C01819=1076.283,415.651,391.048,176.432,32.425,155.839
C01820=1076.291,415.898,391.005,176.438,32.436,155.841
C01821=1076.298,416.143,390.962,176.442,32.446,155.843
C01822=1076.305,416.389,390.920,176.447,32.456,155.846
C01823=1076.313,416.636,390.876,176.453,32.466,155.848
C01824=1076.320,416.882,390.833,176.458,32.477,155.850
C01825=1076.327,417.128,390.790,176.463,32.487,155.853
C01826=1076.334,417.374,390.747,176.469,32.497,155.855
C01827=1076.342,417.620,390.703,176.474,32.507,155.857
C01828=1076.349,417.867,390.660,176.480,32.518,155.859
C01829=1076.356,418.112,390.617,176.485,32.529,155.862
C01830=1076.363,418.358,390.574,176.489,32.539,155.864
C01831=1076.371,418.605,390.530,176.495,32.549,155.867
C01832=1076.378,418.850,390.487,176.500,32.560,155.869
C01833=1076.386,419.097,390.443,176.506,32.571,155.871
C01834=1076.392,419.343,390.400,176.511,32.581,155.874
C01835=1076.400,419.589,390.356,176.517,32.592,155.876
C01836=1076.408,419.835,390.312,176.522,32.602,155.879
C01837=1076.415,420.081,390.269,176.528,32.613,155.881
C01838=1076.423,420.327,390.225,176.533,32.624,155.883
C01839=1076.430,420.573,390.182,176.539,32.635,155.886
C01840=1076.438,420.819,390.139,176.544,32.645,155.888
C01841=1076.446,421.066,390.095,176.550,32.656,155.891
C01842=1076.453,421.311,390.051,176.555,32.667,155.893
C01843=1076.460,421.557,390.007,176.561,32.677,155.896
C01844=1076.468,421.804,389.963,176.566,32.688,155.898
C01845=1076.475,422.049,389.920,176.572,32.700,155.901
C01846=1076.482,422.295,389.875,176.577,32.710,155.903
C01847=1076.490,422.542,389.831,176.583,32.721,155.906
C01848=1076.498,422.787,389.787,176.589,32.733,155.908
C01849=1076.505,423.034,389.743,176.594,32.744,155.911
C01850=1076.513,423.279,389.699,176.600,32.755,155.913
C01851=1076.520,423.525,389.656,176.605,32.766,155.916
C01852=1076.527,423.771,389.611,176.611,32.777,155.918
C01853=1076.535,424.017,389.567,176.617,32.789,155.921
C01854=1076.542,424.263,389.522,176.622,32.800,155.924
C01855=1076.550,424.508,389.478,176.628,32.811,155.926
C01856=1076.557,424.755,389.434,176.634,32.823,155.929
C01857=1076.565,425.001,389.390,176.639,32.834,155.931
C01858=1076.573,425.247,389.345,176.645,32.845,155.934
C01859=1076.580,425.493,389.300,176.651,32.857,155.937
C01860=1076.588,425.738,389.256,176.656,32.868,155.939
C01861=1076.595,425.984,389.212,176.662,32.879,155.942
C01862=1076.604,426.253,389.164,176.668,32.892,155.945
C01863=1076.612,426.521,389.115,176.675,32.905,155.948
C01864=1076.620,426.788,389.066,176.681,32.917,155.951
C01865=1076.629,427.057,389.017,176.687,32.930,155.953
C01866=1076.636,427.303,388.973,176.693,32.942,155.956
C01867=1076.644,427.548,388.928,176.699,32.954,155.959
C01868=1076.652,427.794,388.883,176.705,32.965,155.962
C01869=1076.660,428.040,388.839,176.711,32.977,155.964
C01870=1076.667,428.286,388.794,176.717,32.989,155.967
C01871=1076.674,428.532,388.749,176.723,33.001,155.970
C01872=1076.682,428.778,388.703,176.729,33.013,155.973
C01873=1076.690,429.023,388.659,176.735,33.024,155.975
C01874=1076.697,429.270,388.614,176.740,33.037,155.978
C01875=1076.705,429.515,388.568,176.746,33.048,155.981
C01876=1076.713,429.761,388.524,176.753,33.061,155.984
C01877=1076.721,430.006,388.478,176.759,33.073,155.987
C01878=1076.728,430.252,388.434,176.765,33.085,155.989
C01879=1076.736,430.498,388.388,176.771,33.097,155.992
C01880=1076.744,430.744,388.343,176.777,33.109,155.995
C01881=1076.752,430.989,388.298,176.783,33.122,155.998
C01882=1076.760,431.235,388.252,176.790,33.134,156.001
C01883=1076.767,431.481,388.207,176.796,33.146,156.004
C01884=1076.775,431.726,388.162,176.802,33.159,156.007
C01885=1076.784,431.972,388.116,176.808,33.171,156.010
C01886=1076.791,432.218,388.071,176.814,33.184,156.013
C01887=1076.799,432.464,388.025,176.820,33.196,156.015
C01888=1076.806,432.709,387.980,176.826,33.209,156.018
C01889=1076.814,432.955,387.934,176.832,33.221,156.021
C01890=1076.822,433.201,387.888,176.839,33.234,156.024
C01891=1076.830,433.446,387.842,176.846,33.247,156.027
C01892=1076.837,433.692,387.797,176.852,33.259,156.030
C01893=1076.845,433.937,387.751,176.858,33.272,156.033
C01894=1076.853,434.183,387.705,176.865,33.285,156.036
C01895=1076.861,434.429,387.659,176.871,33.298,156.040
C01896=1076.869,434.673,387.613,176.877,33.311,156.043
C01897=1076.877,434.920,387.567,176.883,33.323,156.046
C01898=1076.885,435.165,387.521,176.890,33.337,156.049
C01899=1076.892,435.410,387.476,176.896,33.349,156.052
C01900=1076.901,435.656,387.429,176.902,33.363,156.055
C01901=1076.909,435.901,387.383,176.910,33.376,156.058
C01902=1076.917,436.147,387.337,176.916,33.389,156.061
C01903=1076.925,436.392,387.291,176.922,33.402,156.064
C01904=1076.932,436.639,387.244,176.929,33.415,156.067
C01905=1076.940,436.884,387.198,176.935,33.429,156.071
C01906=1076.948,437.130,387.152,176.943,33.442,156.074
C01907=1076.956,437.374,387.106,176.949,33.455,156.077
C01908=1076.965,437.620,387.059,176.955,33.468,156.080
C01909=1076.973,437.865,387.013,176.962,33.482,156.083
C01910=1076.981,438.111,386.967,176.969,33.495,156.086
C01911=1076.989,438.356,386.920,176.976,33.509,156.090
C01912=1076.998,438.601,386.873,176.982,33.523,156.093
C01913=1077.005,438.848,386.827,176.988,33.536,156.096
C01914=1077.013,439.093,386.780,176.996,33.550,156.099
C01915=1077.022,439.338,386.734,177.002,33.563,156.103
C01916=1077.030,439.584,386.687,177.009,33.577,156.106
C01917=1077.037,439.829,386.640,177.016,33.591,156.109
C01918=1077.048,440.127,386.582,177.024,33.608,156.113
C01919=1077.057,440.426,386.526,177.033,33.625,156.118
C01920=1077.067,440.725,386.469,177.041,33.642,156.122
C01921=1077.078,441.024,386.411,177.050,33.659,156.126
C01922=1077.086,441.269,386.365,177.056,33.673,156.129
C01923=1077.093,441.515,386.317,177.064,33.688,156.133
C01924=1077.102,441.760,386.270,177.070,33.702,156.136
C01925=1077.110,442.006,386.223,177.078,33.716,156.140
C01926=1077.119,442.250,386.175,177.085,33.730,156.143
C01927=1077.127,442.496,386.128,177.092,33.745,156.147
C01928=1077.135,442.740,386.081,177.099,33.759,156.150
C01929=1077.143,442.986,386.033,177.106,33.773,156.154
C01930=1077.152,443.231,385.986,177.113,33.788,156.157
C01931=1077.159,443.477,385.939,177.121,33.803,156.161
C01932=1077.168,443.722,385.891,177.127,33.817,156.164
C01933=1077.176,443.967,385.843,177.135,33.832,156.168
C01934=1077.185,444.213,385.796,177.143,33.847,156.171
C01935=1077.193,444.458,385.748,177.149,33.861,156.175
C01936=1077.201,444.703,385.700,177.157,33.876,156.179
C01937=1077.210,444.948,385.653,177.164,33.891,156.182
C01938=1077.218,445.193,385.605,177.171,33.906,156.186
C01939=1077.226,445.438,385.557,177.179,33.921,156.190
C01940=1077.235,445.683,385.509,177.186,33.936,156.193
C01941=1077.243,445.928,385.461,177.194,33.951,156.197
C01942=1077.251,446.174,385.413,177.202,33.966,156.201
C01943=1077.259,446.419,385.365,177.209,33.981,156.204
C01944=1077.269,446.664,385.317,177.216,33.996,156.208
C01945=1077.277,446.909,385.269,177.223,34.012,156.212
C01946=1077.285,447.154,385.221,177.230,34.027,156.216
C01947=1077.293,447.399,385.173,177.237,34.042,156.219
C01948=1077.303,447.644,385.124,177.242,34.057,156.223
C01949=1077.311,447.890,385.076,177.248,34.072,156.227
C01950=1077.320,448.134,385.027,177.254,34.087,156.231
C01951=1077.329,448.379,384.980,177.260,34.103,156.235
C01952=1077.337,448.624,384.931,177.265,34.117,156.238
C01953=1077.345,448.869,384.883,177.270,34.133,156.242
C01954=1077.355,449.113,384.836,177.275,34.147,156.246
C01955=1077.367,449.358,384.789,177.280,34.161,156.249
C01956=1077.380,449.603,384.743,177.284,34.174,156.253
C01957=1077.394,449.849,384.697,177.288,34.187,156.256
C01958=1077.034,449.844,384.465,177.267,34.346,156.298
C01959=1077.019,449.599,384.511,177.263,34.333,156.295
C01960=1077.006,449.354,384.556,177.258,34.320,156.291
C01961=1076.995,449.108,384.603,177.253,34.306,156.288
C01962=1076.985,448.864,384.651,177.248,34.292,156.284
C01963=1076.976,448.619,384.698,177.243,34.277,156.280
C01964=1076.967,448.374,384.748,177.237,34.261,156.277
C01965=1076.959,448.130,384.796,177.232,34.246,156.273
C01966=1076.949,447.885,384.844,177.226,34.231,156.269
C01967=1076.941,447.640,384.893,177.220,34.216,156.265
C01968=1076.933,447.395,384.941,177.213,34.201,156.261
C01969=1076.924,447.150,384.990,177.206,34.185,156.258
C01970=1076.916,446.904,385.038,177.199,34.170,156.254
C01971=1076.907,446.660,385.085,177.192,34.156,156.250
C01972=1076.899,446.415,385.134,177.185,34.140,156.246
C01973=1076.891,446.170,385.182,177.177,34.125,156.243
C01974=1076.881,445.924,385.230,177.170,34.110,156.239
C01975=1076.873,445.679,385.278,177.162,34.095,156.235
C01976=1076.865,445.434,385.326,177.155,34.080,156.231
C01977=1076.857,445.189,385.375,177.147,34.065,156.228
C01978=1076.848,444.944,385.422,177.139,34.050,156.224
C01979=1076.840,444.699,385.470,177.132,34.035,156.220
C01980=1076.832,444.453,385.517,177.125,34.020,156.217
C01981=1076.823,444.208,385.565,177.117,34.005,156.213
C01982=1076.815,443.963,385.613,177.110,33.991,156.210
C01983=1076.806,443.718,385.660,177.102,33.976,156.206
C01984=1076.798,443.473,385.708,177.096,33.962,156.202
C01985=1076.789,443.228,385.755,177.088,33.947,156.199
C01986=1076.781,442.982,385.803,177.081,33.932,156.195
C01987=1076.773,442.737,385.851,177.073,33.918,156.192
C01988=1076.765,442.492,385.898,177.067,33.904,156.188
C01989=1076.756,442.246,385.946,177.059,33.889,156.185
C01990=1076.748,442.001,385.993,177.052,33.875,156.181
C01991=1076.740,441.756,386.041,177.045,33.861,156.178
C01992=1076.732,441.511,386.087,177.038,33.847,156.174
C01993=1076.723,441.265,386.134,177.030,33.833,156.171
C01994=1076.715,441.020,386.182,177.024,33.818,156.168
C01995=1076.706,440.739,386.236,177.015,33.802,156.164
C01996=1076.696,440.456,386.289,177.007,33.786,156.160
C01997=1076.687,440.175,386.344,177.000,33.770,156.156
C01998=1076.678,439.894,386.397,176.991,33.754,156.152
C01999=1076.669,439.649,386.444,176.984,33.740,156.149
C02000=1076.661,439.403,386.491,176.978,33.727,156.145
C02001=1076.653,439.158,386.538,176.970,33.713,156.142
C02002=1076.645,438.912,386.584,176.964,33.699,156.139
C02003=1076.636,438.667,386.631,176.957,33.686,156.136
C02004=1076.628,438.421,386.678,176.950,33.672,156.132
C02005=1076.620,438.176,386.725,176.943,33.658,156.129
C02006=1076.612,437.930,386.771,176.937,33.645,156.126
C02007=1076.604,437.685,386.817,176.930,33.631,156.123
C02008=1076.596,437.440,386.864,176.923,33.618,156.119
C02009=1076.587,437.194,386.911,176.916,33.605,156.116
C02010=1076.580,436.949,386.956,176.910,33.591,156.113
C02011=1076.571,436.703,387.003,176.903,33.578,156.110
C02012=1076.564,436.458,387.049,176.896,33.565,156.107
C02013=1076.556,436.212,387.096,176.889,33.552,156.103
C02014=1076.548,435.967,387.142,176.883,33.538,156.100
C02015=1076.539,435.721,387.188,176.877,33.526,156.097
C02016=1076.532,435.476,387.234,176.870,33.513,156.094
C02017=1076.523,435.230,387.281,176.864,33.499,156.091
C02018=1076.516,434.985,387.326,176.857,33.487,156.088
C02019=1076.508,434.739,387.372,176.850,33.473,156.085
C02020=1076.499,434.494,387.419,176.844,33.461,156.082
C02021=1076.492,434.248,387.464,176.837,33.448,156.079
C02022=1076.484,434.003,387.510,176.831,33.435,156.076
C02023=1076.476,433.757,387.556,176.824,33.422,156.073
C02024=1076.468,433.511,387.602,176.818,33.410,156.070
C02025=1076.461,433.266,387.647,176.812,33.397,156.067
C02026=1076.452,433.020,387.693,176.805,33.384,156.064
C02027=1076.445,432.774,387.739,176.799,33.371,156.061
C02028=1076.437,432.529,387.785,176.793,33.359,156.058
C02029=1076.429,432.283,387.830,176.786,33.346,156.055
C02030=1076.421,432.037,387.876,176.780,33.334,156.052
C02031=1076.414,431.792,387.922,176.774,33.321,156.049
C02032=1076.406,431.546,387.968,176.768,33.309,156.046
C02033=1076.398,431.301,388.012,176.761,33.297,156.043
C02034=1076.390,431.055,388.058,176.755,33.285,156.040
C02035=1076.382,430.809,388.104,176.749,33.272,156.037
C02036=1076.375,430.563,388.149,176.742,33.260,156.034
C02037=1076.366,430.318,388.194,176.736,33.248,156.032
C02038=1076.359,430.073,388.239,176.731,33.236,156.029
C02039=1076.351,429.826,388.284,176.725,33.223,156.026
C02040=1076.344,429.581,388.330,176.719,33.211,156.023
C02041=1076.336,429.335,388.374,176.712,33.199,156.020
C02042=1076.328,429.090,388.420,176.706,33.187,156.017
C02043=1076.320,428.843,388.465,176.700,33.176,156.015
C02044=1076.312,428.597,388.509,176.694,33.163,156.012
C02045=1076.304,428.352,388.555,176.688,33.151,156.009
C02046=1076.297,428.106,388.600,176.682,33.140,156.006
C02047=1076.290,427.860,388.645,176.676,33.128,156.004
C02048=1076.282,427.614,388.689,176.670,33.116,156.001
C02049=1076.274,427.368,388.734,176.664,33.104,155.998
C02050=1076.266,427.122,388.779,176.659,33.092,155.995
C02051=1076.258,426.853,388.828,176.651,33.080,155.993
C02052=1076.249,426.583,388.877,176.645,33.067,155.990
C02053=1076.240,426.314,388.926,176.639,33.054,155.987
C02054=1076.232,426.044,388.975,176.632,33.042,155.984
C02055=1076.225,425.798,389.020,176.627,33.031,155.981
C02056=1076.217,425.552,389.064,176.621,33.019,155.978
C02057=1076.210,425.307,389.109,176.615,33.007,155.976
C02058=1076.202,425.061,389.153,176.609,32.996,155.973
C02059=1076.194,424.814,389.197,176.603,32.985,155.970
C02060=1076.187,424.568,389.241,176.597,32.973,155.968
C02061=1076.179,424.323,389.286,176.592,32.962,155.965
C02062=1076.171,424.077,389.331,176.586,32.951,155.963
C02063=1076.164,423.831,389.374,176.580,32.939,155.960
C02064=1076.157,423.585,389.419,176.575,32.929,155.958
C02065=1076.149,423.339,389.463,176.569,32.917,155.955
C02066=1076.141,423.093,389.507,176.564,32.906,155.952
C02067=1076.134,422.847,389.551,176.558,32.895,155.950
C02068=1076.127,422.601,389.595,176.552,32.884,155.947
C02069=1076.119,422.355,389.639,176.547,32.873,155.945
C02070=1076.112,422.109,389.683,176.540,32.862,155.942
C02071=1076.104,421.863,389.727,176.535,32.851,155.940
C02072=1076.096,421.617,389.771,176.529,32.840,155.937
C02073=1076.090,421.371,389.815,176.524,32.829,155.935
C02074=1076.082,421.125,389.859,176.518,32.818,155.932
C02075=1076.074,420.879,389.903,176.513,32.807,155.930
C02076=1076.067,420.634,389.946,176.507,32.797,155.927
C02077=1076.059,420.387,389.990,176.502,32.786,155.925
C02078=1076.051,420.141,390.033,176.496,32.775,155.923
C02079=1076.044,419.895,390.077,176.491,32.764,155.920
C02080=1076.037,419.648,390.121,176.485,32.754,155.918
C02081=1076.030,419.403,390.164,176.480,32.743,155.915
C02082=1076.022,419.156,390.208,176.474,32.733,155.913
C02083=1076.014,418.910,390.251,176.469,32.722,155.911
C02084=1076.007,418.664,390.295,176.463,32.711,155.908
C02085=1076.000,418.418,390.338,176.458,32.701,155.906
C02086=1075.992,418.172,390.382,176.453,32.691,155.903
C02087=1075.985,417.926,390.425,176.447,32.680,155.901
C02088=1075.977,417.680,390.468,176.442,32.670,155.899
C02089=1075.970,417.434,390.512,176.436,32.660,155.896
C02090=1075.963,417.188,390.555,176.431,32.649,155.894
C02091=1075.956,416.942,390.598,176.426,32.639,155.892
C02092=1075.948,416.696,390.641,176.421,32.628,155.889
C02093=1075.941,416.450,390.685,176.416,32.618,155.887
C02094=1075.933,416.203,390.728,176.411,32.608,155.885
C02095=1075.926,415.957,390.771,176.405,32.598,155.882
C02096=1075.919,415.712,390.814,176.400,32.587,155.880
C02097=1075.911,415.465,390.857,176.395,32.578,155.878
C02098=1075.904,415.219,390.900,176.389,32.567,155.876
C02099=1075.897,414.973,390.943,176.384,32.557,155.873
C02100=1075.890,414.726,390.986,176.379,32.547,155.871
C02101=1075.882,414.480,391.028,176.374,32.537,155.869
C02102=1075.875,414.234,391.071,176.368,32.527,155.867
C02103=1075.867,413.988,391.115,176.363,32.517,155.864
C02104=1075.861,413.741,391.157,176.358,32.507,155.862
C02105=1075.853,413.495,391.199,176.354,32.497,155.860
C02106=1075.845,413.249,391.243,176.348,32.487,155.858
C02107=1075.838,412.997,391.286,176.343,32.478,155.856
C02108=1075.831,412.745,391.329,176.338,32.468,155.853
C02109=1075.823,412.493,391.373,176.332,32.458,155.851
C02110=1075.816,412.241,391.417,176.327,32.448,155.849
C02111=1075.809,411.995,391.459,176.322,32.438,155.847
C02112=1075.801,411.749,391.501,176.317,32.429,155.845
C02113=1075.794,411.502,391.544,176.312,32.419,155.842
C02114=1075.787,411.255,391.587,176.307,32.409,155.840
C02115=1075.779,411.010,391.629,176.302,32.399,155.838
C02116=1075.773,410.763,391.671,176.297,32.390,155.836
C02117=1075.766,410.517,391.714,176.292,32.380,155.834
C02118=1075.758,410.271,391.756,176.287,32.371,155.832
C02119=1075.751,410.025,391.798,176.282,32.361,155.830
C02120=1075.744,409.778,391.841,176.277,32.352,155.828
C02121=1075.736,409.532,391.883,176.272,32.342,155.826
C02122=1075.730,409.285,391.925,176.267,32.333,155.823
C02123=1075.722,409.039,391.967,176.262,32.323,155.821
C02124=1075.715,408.793,392.009,176.257,32.314,155.819
C02125=1075.708,408.546,392.052,176.252,32.305,155.817
C02126=1075.701,408.300,392.093,176.247,32.295,155.815
C02127=1075.694,408.053,392.136,176.243,32.286,155.813
C02128=1075.687,407.807,392.178,176.238,32.276,155.811
C02129=1075.680,407.561,392.219,176.233,32.268,155.809
C02130=1075.673,407.314,392.262,176.228,32.258,155.807
C02131=1075.667,407.068,392.303,176.223,32.249,155.805
C02132=1075.660,406.822,392.345,176.219,32.240,155.803
C02133=1075.652,406.575,392.387,176.214,32.230,155.801
C02134=1075.645,406.329,392.429,176.209,32.221,155.799
C02135=1075.638,406.083,392.470,176.204,32.213,155.797
C02136=1075.631,405.837,392.512,176.199,32.203,155.795
C02137=1075.624,405.590,392.554,176.195,32.194,155.793
C02138=1075.617,405.343,392.595,176.190,32.185,155.791
C02139=1075.609,405.097,392.637,176.185,32.176,155.789
C02140=1075.603,404.850,392.679,176.180,32.167,155.787
C02141=1075.595,404.604,392.720,176.175,32.158,155.785
C02142=1075.589,404.358,392.761,176.171,32.149,155.783
C02143=1075.582,404.111,392.804,176.166,32.141,155.781
C02144=1075.575,403.865,392.845,176.162,32.132,155.779
C02145=1075.567,403.618,392.886,176.157,32.123,155.777
C02146=1075.560,403.372,392.927,176.152,32.114,155.775
C02147=1075.554,403.125,392.969,176.148,32.105,155.774
C02148=1075.547,402.879,393.010,176.143,32.096,155.772
C02149=1075.539,402.632,393.051,176.138,32.088,155.770
C02150=1075.532,402.386,393.093,176.133,32.079,155.768
C02151=1075.525,402.139,393.134,176.129,32.070,155.766
C02152=1075.518,401.893,393.175,176.124,32.062,155.764
C02153=1075.512,401.646,393.216,176.120,32.053,155.762
C02154=1075.504,401.400,393.258,176.115,32.044,155.760
C02155=1075.498,401.154,393.299,176.111,32.035,155.759
C02156=1075.490,400.907,393.340,176.106,32.027,155.757
C02157=1075.483,400.661,393.381,176.101,32.019,155.755
C02158=1075.477,400.414,393.421,176.096,32.010,155.753
C02159=1075.470,400.179,393.461,176.093,32.002,155.751
C02160=1075.464,399.943,393.500,176.088,31.994,155.750
C02161=1075.456,399.708,393.539,176.084,31.986,155.748
C02162=1075.450,399.472,393.578,176.079,31.978,155.746
C02163=1075.443,399.237,393.618,176.075,31.970,155.744
C02164=1075.437,399.001,393.657,176.071,31.961,155.743
C02165=1075.430,398.765,393.695,176.066,31.953,155.741
C02166=1075.421,398.432,393.750,176.060,31.942,155.738
C02167=1075.414,398.186,393.791,176.056,31.934,155.737
C02168=1075.407,397.939,393.832,176.051,31.925,155.735
C02169=1075.400,397.692,393.873,176.047,31.917,155.733
C02170=1075.393,397.446,393.913,176.043,31.909,155.731
C02171=1075.386,397.199,393.954,176.038,31.901,155.730
C02172=1075.380,396.953,393.994,176.033,31.892,155.728
C02173=1075.372,396.706,394.036,176.029,31.885,155.726
C02174=1075.366,396.460,394.076,176.025,31.876,155.724
C02175=1075.358,396.213,394.116,176.020,31.868,155.723
C02176=1075.351,395.967,394.157,176.015,31.860,155.721
C02177=1075.345,395.720,394.197,176.012,31.852,155.719
C02178=1075.338,395.473,394.237,176.007,31.844,155.717
C02179=1075.331,395.227,394.278,176.002,31.835,155.716
C02180=1075.324,394.980,394.319,175.998,31.827,155.714
C02181=1075.317,394.734,394.358,175.994,31.819,155.712
C02182=1075.311,394.487,394.398,175.989,31.811,155.711
C02183=1075.304,394.240,394.439,175.985,31.803,155.709
C02184=1075.297,393.994,394.480,175.981,31.795,155.707
C02185=1075.290,393.747,394.520,175.976,31.787,155.705
C02186=1075.283,393.501,394.560,175.972,31.779,155.704
C02187=1075.277,393.254,394.600,175.968,31.772,155.702
C02188=1075.269,393.007,394.640,175.963,31.764,155.701
C02189=1075.263,392.761,394.680,175.959,31.756,155.699
C02190=1075.256,392.514,394.720,175.954,31.748,155.697
C02191=1075.249,392.268,394.760,175.950,31.740,155.695
C02192=1075.242,392.021,394.800,175.946,31.732,155.694
C02193=1075.236,391.774,394.840,175.941,31.724,155.692
C02194=1075.229,391.528,394.880,175.937,31.716,155.691
C02195=1075.222,391.282,394.920,175.933,31.709,155.689
C02196=1075.215,391.034,394.959,175.928,31.701,155.687
C02197=1075.208,390.788,394.999,175.924,31.694,155.686
C02198=1075.201,390.541,395.039,175.920,31.686,155.684
C02199=1075.195,390.295,395.079,175.915,31.678,155.683
C02200=1075.187,390.048,395.119,175.912,31.670,155.681
C02201=1075.181,389.801,395.158,175.907,31.663,155.679
C02202=1075.174,389.555,395.198,175.902,31.655,155.678
C02203=1075.167,389.308,395.237,175.899,31.648,155.676
C02204=1075.161,389.061,395.277,175.894,31.640,155.675
C02205=1075.153,388.814,395.317,175.890,31.633,155.673
C02206=1075.147,388.568,395.357,175.886,31.625,155.671
C02207=1075.140,388.321,395.396,175.881,31.617,155.670
C02208=1075.133,388.075,395.435,175.877,31.610,155.668
C02209=1075.127,387.828,395.475,175.873,31.603,155.667
C02210=1075.120,387.582,395.514,175.869,31.595,155.665
C02211=1075.113,387.335,395.553,175.864,31.588,155.664
C02212=1075.106,387.088,395.593,175.861,31.580,155.662
C02213=1075.100,386.841,395.632,175.856,31.573,155.661
C02214=1075.093,386.595,395.672,175.852,31.565,155.659
C02215=1075.086,386.354,395.710,175.848,31.558,155.658
C02216=1075.080,386.114,395.748,175.844,31.551,155.656
C02217=1075.074,385.874,395.786,175.839,31.544,155.655
C02218=1075.067,385.633,395.825,175.836,31.537,155.653
C02219=1075.060,385.394,395.863,175.832,31.530,155.652
C02220=1075.054,385.153,395.901,175.828,31.522,155.650
C02221=1075.047,384.913,395.940,175.824,31.515,155.649
C02222=1075.041,384.672,395.978,175.819,31.508,155.647
C02223=1075.034,384.425,396.017,175.816,31.501,155.646
C02224=1075.027,384.179,396.056,175.811,31.494,155.644
C02225=1075.021,383.932,396.095,175.807,31.486,155.643
C02226=1075.015,383.686,396.134,175.804,31.479,155.641
C02227=1075.008,383.439,396.173,175.799,31.472,155.640
C02228=1075.001,383.192,396.212,175.795,31.464,155.638
C02229=1074.995,382.945,396.251,175.791,31.457,155.637
C02230=1074.988,382.698,396.290,175.787,31.451,155.635
C02231=1074.981,382.451,396.329,175.782,31.443,155.634
C02232=1074.974,382.204,396.368,175.779,31.436,155.632
C02233=1074.968,381.957,396.407,175.774,31.429,155.631
C02234=1074.962,381.711,396.445,175.771,31.422,155.629
C02235=1074.955,381.464,396.484,175.766,31.415,155.628
C02236=1074.949,381.218,396.523,175.762,31.408,155.627
C02237=1074.942,380.971,396.562,175.759,31.401,155.625
C02238=1074.935,380.724,396.601,175.754,31.394,155.624
C02239=1074.928,380.477,396.640,175.750,31.387,155.622
C02240=1074.922,380.230,396.678,175.746,31.380,155.621
C02241=1074.915,379.983,396.717,175.742,31.373,155.619
C02242=1074.909,379.737,396.755,175.739,31.366,155.618
C02243=1074.902,379.490,396.794,175.734,31.359,155.617
C02244=1074.895,379.243,396.831,175.730,31.352,155.615
C02245=1074.888,378.996,396.870,175.726,31.345,155.614
C02246=1074.881,378.749,396.909,175.722,31.338,155.612
C02247=1074.875,378.502,396.947,175.719,31.332,155.611
C02248=1074.868,378.256,396.986,175.714,31.324,155.610
C02249=1074.862,378.008,397.024,175.710,31.318,155.608
C02250=1074.855,377.761,397.063,175.706,31.311,155.607
C02251=1074.849,377.515,397.101,175.702,31.304,155.605
C02252=1074.842,377.268,397.139,175.698,31.298,155.604
C02253=1074.835,377.021,397.178,175.694,31.291,155.603
C02254=1074.829,376.773,397.216,175.690,31.284,155.601
C02255=1074.823,376.527,397.255,175.687,31.277,155.600
C02256=1074.815,376.280,397.292,175.682,31.270,155.599
C02257=1074.809,376.033,397.330,175.678,31.264,155.597
C02258=1074.803,375.787,397.369,175.675,31.257,155.596
C02259=1074.796,375.539,397.407,175.670,31.250,155.595
C02260=1074.789,375.292,397.446,175.667,31.243,155.593
C02261=1074.783,375.046,397.484,175.663,31.237,155.592
C02262=1074.777,374.798,397.522,175.658,31.230,155.590
C02263=1074.771,374.551,397.559,175.655,31.223,155.589
C02264=1074.764,374.305,397.598,175.651,31.217,155.588
C02265=1074.757,374.057,397.636,175.648,31.210,155.586
C02266=1074.751,373.811,397.674,175.643,31.203,155.585
C02267=1074.745,373.563,397.712,175.639,31.197,155.584
C02268=1074.738,373.317,397.750,175.636,31.191,155.583
C02269=1074.731,373.070,397.788,175.631,31.183,155.581
C02270=1074.725,372.823,397.826,175.628,31.177,155.580
C02271=1074.718,372.597,397.860,175.624,31.171,155.579
C02272=1074.713,372.371,397.895,175.620,31.165,155.578
C02273=1074.707,372.145,397.928,175.617,31.159,155.576
C02274=1074.701,371.920,397.963,175.613,31.153,155.575
C02275=1074.695,371.694,397.998,175.610,31.148,155.574
C02276=1074.689,371.468,398.032,175.607,31.142,155.573
C02277=1074.683,371.243,398.067,175.603,31.136,155.572
C02278=1074.677,371.017,398.102,175.600,31.130,155.570
C02279=1074.670,370.770,398.139,175.596,31.124,155.569
C02280=1074.664,370.523,398.177,175.591,31.117,155.568
C02281=1074.657,370.276,398.213,175.588,31.111,155.567
C02282=1074.651,370.028,398.252,175.584,31.104,155.565
C02283=1074.644,369.782,398.289,175.581,31.098,155.564
C02284=1074.638,369.535,398.327,175.576,31.092,155.563
C02285=1074.631,369.288,398.364,175.572,31.086,155.562
C02286=1074.625,369.041,398.402,175.569,31.079,155.560
C02287=1074.618,368.794,398.439,175.565,31.073,155.559
C02288=1074.612,368.546,398.477,175.562,31.067,155.558
C02289=1074.605,368.300,398.514,175.557,31.060,155.557
C02290=1074.600,368.052,398.551,175.554,31.054,155.555
C02291=1074.592,367.805,398.588,175.550,31.048,155.554
C02292=1074.586,367.559,398.626,175.546,31.041,155.553
C02293=1074.579,367.311,398.663,175.543,31.035,155.552
C02294=1074.574,367.064,398.701,175.538,31.029,155.550
C02295=1074.567,366.818,398.738,175.535,31.023,155.549
C02296=1074.561,366.570,398.775,175.531,31.016,155.548
C02297=1074.554,366.323,398.812,175.527,31.010,155.547
C02298=1074.548,366.076,398.849,175.524,31.004,155.546
C02299=1074.541,365.829,398.887,175.519,30.998,155.544
C02300=1074.536,365.581,398.924,175.516,30.992,155.543
C02301=1074.529,365.335,398.961,175.512,30.985,155.542
C02302=1074.522,365.087,398.998,175.509,30.979,155.541
C02303=1074.516,364.840,399.036,175.505,30.973,155.540
C02304=1074.510,364.593,399.072,175.501,30.967,155.538
C02305=1074.503,364.345,399.109,175.498,30.961,155.537
C02306=1074.497,364.099,399.147,175.493,30.955,155.536
C02307=1074.491,363.852,399.183,175.490,30.949,155.535
C02308=1074.484,363.604,399.220,175.486,30.943,155.534
C02309=1074.477,363.357,399.257,175.483,30.937,155.532
C02310=1074.471,363.110,399.294,175.479,30.931,155.531
C02311=1074.465,362.862,399.331,175.475,30.925,155.530
C02312=1074.458,362.615,399.368,175.472,30.919,155.529
C02313=1074.452,362.368,399.404,175.467,30.913,155.528
C02314=1074.445,362.122,399.441,175.464,30.907,155.527
C02315=1074.438,361.874,399.478,175.460,30.901,155.525
C02316=1074.433,361.627,399.515,175.457,30.895,155.524
C02317=1074.426,361.380,399.551,175.453,30.889,155.523
C02318=1074.420,361.133,399.588,175.449,30.883,155.522
C02319=1074.413,360.885,399.625,175.446,30.877,155.521
C02320=1074.407,360.638,399.661,175.442,30.871,155.520
C02321=1074.400,360.391,399.698,175.439,30.865,155.518
C02322=1074.394,360.144,399.734,175.434,30.859,155.517
C02323=1074.388,359.896,399.771,175.431,30.853,155.516
C02324=1074.382,359.649,399.807,175.427,30.848,155.515
C02325=1074.375,359.401,399.844,175.424,30.842,155.514
C02326=1074.369,359.154,399.881,175.420,30.836,155.513
C02327=1074.363,358.937,399.912,175.417,30.831,155.512
C02328=1074.357,358.720,399.945,175.414,30.826,155.511
C02329=1074.352,358.503,399.976,175.410,30.821,155.510
C02330=1074.346,358.285,400.009,175.407,30.815,155.509
C02331=1074.340,358.068,400.040,175.404,30.810,155.508
C02332=1074.335,357.850,400.072,175.401,30.805,155.507
C02333=1074.329,357.633,400.105,175.398,30.800,155.506
C02334=1074.324,357.416,400.137,175.395,30.795,155.505
C02335=1074.317,357.168,400.173,175.391,30.790,155.504
C02336=1074.311,356.921,400.209,175.387,30.783,155.503
C02337=1074.305,356.674,400.246,175.383,30.778,155.502
C02338=1074.298,356.426,400.282,175.380,30.772,155.501
C02339=1074.292,356.179,400.318,175.376,30.766,155.499
C02340=1074.285,355.932,400.354,175.373,30.760,155.498
C02341=1074.279,355.685,400.390,175.369,30.755,155.497
C02342=1074.273,355.437,400.426,175.366,30.750,155.496
C02343=1074.267,355.190,400.462,175.362,30.744,155.495
C02344=1074.260,354.943,400.499,175.358,30.738,155.494
C02345=1074.254,354.696,400.534,175.355,30.732,155.493
C02346=1074.248,354.448,400.571,175.351,30.727,155.492
C02347=1074.242,354.201,400.607,175.348,30.721,155.491
C02348=1074.236,353.954,400.643,175.344,30.715,155.490
C02349=1074.229,353.706,400.678,175.341,30.710,155.489
C02350=1074.222,353.459,400.715,175.337,30.704,155.488
C02351=1074.216,353.212,400.750,175.334,30.698,155.486
C02352=1074.210,352.965,400.787,175.330,30.693,155.485
C02353=1074.204,352.717,400.823,175.326,30.687,155.484
C02354=1074.198,352.469,400.858,175.323,30.682,155.483
C02355=1074.191,352.223,400.894,175.319,30.676,155.482
C02356=1074.185,351.975,400.930,175.316,30.670,155.481
C02357=1074.179,351.727,400.966,175.312,30.665,155.480
C02358=1074.172,351.480,401.001,175.309,30.659,155.479
C02359=1074.166,351.233,401.037,175.305,30.654,155.478
C02360=1074.160,350.985,401.073,175.302,30.648,155.477
C02361=1074.153,350.738,401.108,175.298,30.643,155.476
C02362=1074.147,350.491,401.144,175.295,30.638,155.475
C02363=1074.141,350.243,401.180,175.292,30.632,155.474
C02364=1074.134,349.996,401.215,175.288,30.627,155.473
C02365=1074.128,349.749,401.251,175.285,30.621,155.472
C02366=1074.122,349.501,401.286,175.281,30.616,155.471
C02367=1074.116,349.254,401.322,175.278,30.610,155.470
C02368=1074.109,349.007,401.358,175.274,30.605,155.469
C02369=1074.102,348.759,401.393,175.271,30.600,155.468
C02370=1074.096,348.511,401.429,175.267,30.594,155.467
C02371=1074.091,348.265,401.464,175.264,30.589,155.466
C02372=1074.084,348.017,401.499,175.260,30.583,155.465
C02373=1074.078,347.769,401.535,175.256,30.578,155.464
C02374=1074.071,347.522,401.570,175.253,30.572,155.463
C02375=1074.065,347.274,401.606,175.249,30.567,155.462
C02376=1074.059,347.027,401.641,175.247,30.562,155.461
C02377=1074.053,346.780,401.676,175.243,30.556,155.460
C02378=1074.046,346.533,401.712,175.240,30.551,155.459
C02379=1074.041,346.284,401.747,175.236,30.545,155.458
C02380=1074.035,346.037,401.782,175.233,30.540,155.457
C02381=1074.029,345.790,401.817,175.229,30.535,155.456
C02382=1074.022,345.543,401.852,175.226,30.529,155.455
C02383=1074.017,345.327,401.883,175.223,30.525,155.454
C02384=1074.011,345.112,401.914,175.219,30.520,155.453
C02385=1074.005,344.896,401.944,175.217,30.516,155.452
C02386=1074.001,344.680,401.975,175.214,30.511,155.451
C02387=1073.995,344.464,402.006,175.211,30.506,155.450
C02388=1073.989,344.249,402.037,175.208,30.502,155.449
C02389=1073.984,344.033,402.067,175.205,30.497,155.449
C02390=1073.979,343.817,402.098,175.202,30.492,155.448
C02391=1073.972,343.570,402.133,175.198,30.487,155.447
C02392=1073.966,343.321,402.168,175.195,30.482,155.446
C02393=1073.960,343.075,402.203,175.192,30.477,155.445
C02394=1073.953,342.827,402.238,175.189,30.472,155.444
C02395=1073.947,342.579,402.272,175.185,30.467,155.443
C02396=1073.941,342.332,402.307,175.181,30.462,155.442
C02397=1073.935,342.084,402.342,175.178,30.456,155.441
C02398=1073.928,341.837,402.377,175.174,30.451,155.440
C02399=1073.922,341.590,402.411,175.171,30.446,155.439
C02400=1073.916,341.342,402.447,175.168,30.441,155.438
C02401=1073.910,341.094,402.481,175.165,30.436,155.437
C02402=1073.904,340.848,402.516,175.161,30.430,155.436
C02403=1073.897,340.600,402.550,175.158,30.425,155.435
C02404=1073.891,340.352,402.586,175.154,30.420,155.434
C02405=1073.885,340.105,402.620,175.152,30.415,155.433
C02406=1073.879,339.857,402.655,175.148,30.410,155.432
C02407=1073.873,339.610,402.689,175.145,30.405,155.432
C02408=1073.867,339.362,402.724,175.141,30.399,155.431
C02409=1073.860,339.114,402.760,175.137,30.394,155.430
C02410=1073.854,338.867,402.794,175.134,30.389,155.429
C02411=1073.848,338.620,402.829,175.131,30.384,155.428
C02412=1073.842,338.372,402.863,175.128,30.379,155.427
C02413=1073.836,338.124,402.898,175.124,30.374,155.426
C02414=1073.830,337.877,402.932,175.121,30.369,155.425
C02415=1073.823,337.629,402.967,175.118,30.364,155.424
C02416=1073.817,337.382,403.001,175.115,30.359,155.423
C02417=1073.811,337.134,403.035,175.111,30.354,155.422
C02418=1073.805,336.886,403.070,175.108,30.349,155.421
C02419=1073.799,336.639,403.104,175.104,30.344,155.420
C02420=1073.792,336.391,403.138,175.102,30.339,155.419
C02421=1073.786,336.144,403.173,175.098,30.334,155.418
C02422=1073.780,335.896,403.208,175.095,30.329,155.418
C02423=1073.774,335.649,403.242,175.091,30.324,155.417
C02424=1073.767,335.401,403.276,175.088,30.319,155.416
C02425=1073.761,335.154,403.310,175.085,30.314,155.415
C02426=1073.755,334.906,403.344,175.081,30.309,155.414
C02427=1073.749,334.658,403.379,175.078,30.304,155.413
C02428=1073.743,334.410,403.413,175.075,30.299,155.412
C02429=1073.737,334.163,403.447,175.072,30.294,155.411
C02430=1073.731,333.916,403.481,175.068,30.289,155.410
C02431=1073.724,333.668,403.515,175.065,30.284,155.409
C02432=1073.719,333.421,403.550,175.062,30.279,155.409
C02433=1073.712,333.173,403.584,175.059,30.274,155.408
C02434=1073.706,332.925,403.618,175.055,30.269,155.407
C02435=1073.700,332.677,403.652,175.052,30.264,155.406
C02436=1073.693,332.430,403.685,175.049,30.260,155.405
C02437=1073.688,332.182,403.719,175.046,30.255,155.404
C02438=1073.681,331.934,403.754,175.042,30.250,155.403
C02439=1073.676,331.716,403.783,175.039,30.245,155.402
C02440=1073.671,331.498,403.814,175.037,30.241,155.402
C02441=1073.666,331.280,403.844,175.034,30.237,155.401
C02442=1073.660,331.062,403.874,175.031,30.232,155.400
C02443=1073.655,330.844,403.904,175.028,30.228,155.399
C02444=1073.649,330.625,403.933,175.025,30.224,155.399
C02445=1073.643,330.407,403.963,175.022,30.219,155.398
C02446=1073.638,330.189,403.992,175.019,30.216,155.397
C02447=1073.631,329.940,404.026,175.016,30.211,155.396
C02448=1073.625,329.693,404.060,175.013,30.206,155.395
C02449=1073.618,329.445,404.094,175.010,30.201,155.395
C02450=1073.613,329.198,404.127,175.006,30.196,155.394
C02451=1073.606,328.951,404.161,175.004,30.192,155.393
C02452=1073.600,328.703,404.195,175.000,30.187,155.392
C02453=1073.593,328.455,404.228,174.997,30.182,155.391
C02454=1073.588,328.208,404.262,174.994,30.178,155.390
C02455=1073.581,327.959,404.295,174.990,30.172,155.389
C02456=1073.575,327.712,404.329,174.987,30.168,155.389
C02457=1073.569,327.464,404.363,174.984,30.163,155.388
C02458=1073.562,327.217,404.396,174.981,30.159,155.387
C02459=1073.557,326.969,404.430,174.977,30.154,155.386
C02460=1073.550,326.722,404.463,174.975,30.149,155.385
C02461=1073.544,326.474,404.497,174.971,30.144,155.384
C02462=1073.538,326.225,404.530,174.968,30.140,155.384
C02463=1073.532,325.978,404.564,174.965,30.135,155.383
C02464=1073.525,325.731,404.596,174.962,30.130,155.382
C02465=1073.519,325.483,404.631,174.958,30.126,155.381
C02466=1073.513,325.235,404.664,174.956,30.121,155.380
C02467=1073.507,324.987,404.697,174.952,30.116,155.379
C02468=1073.500,324.740,404.730,174.950,30.111,155.378
C02469=1073.495,324.492,404.764,174.946,30.107,155.378
C02470=1073.488,324.244,404.797,174.943,30.102,155.377
C02471=1073.482,323.996,404.830,174.940,30.098,155.376
C02472=1073.476,323.749,404.864,174.936,30.093,155.375
C02473=1073.470,323.501,404.897,174.933,30.088,155.374
C02474=1073.464,323.254,404.930,174.930,30.084,155.374
C02475=1073.458,323.006,404.963,174.927,30.079,155.373
C02476=1073.451,322.758,404.997,174.924,30.074,155.372
C02477=1073.446,322.510,405.030,174.921,30.070,155.371
C02478=1073.439,322.262,405.063,174.917,30.065,155.370
C02479=1073.434,322.015,405.096,174.915,30.060,155.369
C02480=1073.428,321.767,405.129,174.911,30.055,155.368
C02481=1073.421,321.519,405.162,174.909,30.051,155.368
C02482=1073.416,321.271,405.195,174.905,30.046,155.367
C02483=1073.409,321.024,405.228,174.902,30.041,155.366
C02484=1073.404,320.777,405.262,174.899,30.037,155.365
C02485=1073.397,320.529,405.295,174.896,30.032,155.364
C02486=1073.392,320.281,405.328,174.893,30.027,155.364
C02487=1073.385,320.033,405.361,174.890,30.023,155.363
C02488=1073.379,319.785,405.394,174.887,30.019,155.362
C02489=1073.373,319.537,405.427,174.884,30.013,155.361
C02490=1073.367,319.290,405.460,174.880,30.009,155.360
C02491=1073.361,319.042,405.493,174.877,30.005,155.360
C02492=1073.355,318.794,405.525,174.874,30.000,155.359
C02493=1073.349,318.546,405.558,174.871,29.995,155.358
C02494=1073.343,318.298,405.591,174.868,29.991,155.357
C02495=1073.338,318.077,405.620,174.865,29.986,155.356
C02496=1073.333,317.856,405.651,174.863,29.982,155.356
C02497=1073.328,317.634,405.679,174.860,29.978,155.355
C02498=1073.322,317.413,405.709,174.858,29.974,155.354
C02499=1073.317,317.192,405.738,174.854,29.970,155.354
C02500=1073.311,316.970,405.767,174.852,29.966,155.353
C02501=1073.306,316.749,405.797,174.849,29.962,155.352
C02502=1073.300,316.527,405.826,174.846,29.958,155.351
C02503=1073.295,316.280,405.859,174.843,29.953,155.350
C02504=1073.289,316.031,405.891,174.840,29.949,155.350
C02505=1073.283,315.784,405.924,174.837,29.944,155.349
C02506=1073.278,315.537,405.957,174.834,29.939,155.348
C02507=1073.272,315.288,405.989,174.831,29.935,155.347
C02508=1073.265,315.041,406.022,174.828,29.930,155.346
C02509=1073.260,314.793,406.055,174.825,29.926,155.346
C02510=1073.254,314.545,406.088,174.822,29.921,155.345
C02511=1073.248,314.297,406.120,174.819,29.916,155.344
C02512=1073.241,314.049,406.153,174.816,29.912,155.343
C02513=1073.235,313.801,406.185,174.813,29.908,155.343
C02514=1073.229,313.554,406.218,174.810,29.904,155.342
C02515=1073.223,313.305,406.250,174.807,29.899,155.341
C02516=1073.216,313.058,406.282,174.804,29.895,155.340
C02517=1073.210,312.810,406.314,174.801,29.890,155.339
C02518=1073.204,312.563,406.346,174.798,29.886,155.339
C02519=1073.198,312.315,406.378,174.795,29.881,155.338
C02520=1073.192,312.067,406.411,174.792,29.877,155.337
C02521=1073.186,311.819,406.443,174.788,29.873,155.336
C02522=1073.180,311.571,406.476,174.786,29.868,155.336
C02523=1073.173,311.323,406.507,174.782,29.864,155.335
C02524=1073.167,311.076,406.540,174.780,29.860,155.334
C02525=1073.161,310.828,406.572,174.776,29.855,155.333
C02526=1073.155,310.579,406.604,174.774,29.851,155.333
C02527=1073.149,310.333,406.636,174.770,29.847,155.332
C02528=1073.143,310.084,406.668,174.768,29.842,155.331
C02529=1073.136,309.836,406.700,174.764,29.838,155.330
C02530=1073.130,309.589,406.732,174.762,29.833,155.330
C02531=1073.124,309.341,406.764,174.758,29.829,155.329
C02532=1073.119,309.093,406.796,174.756,29.825,155.328
C02533=1073.112,308.846,406.829,174.752,29.820,155.327
C02534=1073.106,308.598,406.860,174.750,29.816,155.327
C02535=1073.100,308.349,406.892,174.746,29.811,155.326
C02536=1073.094,308.101,406.924,174.744,29.807,155.325
C02537=1073.088,307.854,406.957,174.740,29.803,155.324
C02538=1073.082,307.606,406.989,174.738,29.798,155.324
C02539=1073.075,307.358,407.020,174.735,29.794,155.323
C02540=1073.070,307.111,407.052,174.732,29.790,155.322
C02541=1073.064,306.862,407.084,174.729,29.786,155.321
C02542=1073.058,306.614,407.116,174.726,29.781,155.321
C02543=1073.051,306.367,407.148,174.723,29.777,155.320
C02544=1073.045,306.119,407.180,174.720,29.772,155.319
C02545=1073.040,305.871,407.212,174.717,29.768,155.318
C02546=1073.034,305.623,407.244,174.714,29.764,155.318
C02547=1073.027,305.376,407.275,174.711,29.759,155.317
C02548=1073.021,305.128,407.307,174.709,29.755,155.316
C02549=1073.015,304.879,407.339,174.705,29.751,155.315
C02550=1073.009,304.632,407.370,174.702,29.746,155.315
C02551=1073.004,304.412,407.399,174.700,29.743,155.314
C02552=1072.999,304.193,407.427,174.697,29.739,155.313
C02553=1072.993,303.973,407.455,174.695,29.735,155.313
C02554=1072.988,303.753,407.482,174.692,29.731,155.312
C02555=1072.983,303.533,407.511,174.689,29.727,155.311
C02556=1072.978,303.314,407.539,174.686,29.723,155.311
C02557=1072.973,303.094,407.567,174.684,29.719,155.310
C02558=1072.967,302.874,407.595,174.681,29.715,155.309
C02559=1072.961,302.626,407.627,174.678,29.711,155.309
C02560=1072.955,302.378,407.658,174.676,29.707,155.308
C02561=1072.949,302.130,407.690,174.672,29.703,155.307
C02562=1072.944,301.882,407.721,174.670,29.698,155.306
C02563=1072.937,301.635,407.753,174.666,29.694,155.306
C02564=1072.932,301.387,407.784,174.664,29.690,155.305
C02565=1072.926,301.139,407.816,174.661,29.685,155.304
C02566=1072.920,300.891,407.847,174.658,29.681,155.303
C02567=1072.914,300.643,407.879,174.655,29.677,155.303
C02568=1072.909,300.395,407.910,174.652,29.672,155.302
C02569=1072.902,300.147,407.942,174.649,29.668,155.301
C02570=1072.897,299.899,407.973,174.647,29.664,155.301
C02571=1072.890,299.651,408.004,174.643,29.659,155.300
C02572=1072.885,299.404,408.036,174.641,29.655,155.299
C02573=1072.879,299.155,408.067,174.638,29.651,155.298
C02574=1072.873,298.908,408.098,174.635,29.647,155.298
C02575=1072.867,298.660,408.130,174.632,29.642,155.297
C02576=1072.862,298.411,408.161,174.630,29.638,155.296
C02577=1072.856,298.164,408.192,174.626,29.634,155.295
C02578=1072.850,297.916,408.224,174.624,29.629,155.295
C02579=1072.844,297.668,408.255,174.621,29.625,155.294
C02580=1072.838,297.420,408.287,174.618,29.621,155.293
C02581=1072.832,297.172,408.317,174.615,29.616,155.292
C02582=1072.826,296.924,408.349,174.612,29.612,155.292
C02583=1072.820,296.676,408.379,174.609,29.608,155.291
C02584=1072.814,296.428,408.411,174.607,29.604,155.290
C02585=1072.809,296.180,408.442,174.603,29.599,155.290
C02586=1072.802,295.932,408.473,174.601,29.596,155.289
C02587=1072.796,295.684,408.504,174.598,29.591,155.288
C02588=1072.791,295.437,408.535,174.595,29.587,155.287
C02589=1072.784,295.188,408.566,174.592,29.583,155.287
C02590=1072.779,294.941,408.596,174.590,29.579,155.286
C02591=1072.773,294.692,408.628,174.586,29.575,155.285
C02592=1072.767,294.445,408.659,174.584,29.570,155.285
C02593=1072.760,294.197,408.690,174.581,29.566,155.284
C02594=1072.754,293.949,408.721,174.578,29.562,155.283
C02595=1072.748,293.701,408.751,174.575,29.558,155.283
C02596=1072.743,293.452,408.782,174.573,29.553,155.282
C02597=1072.737,293.205,408.813,174.569,29.549,155.281
C02598=1072.730,292.956,408.844,174.567,29.546,155.280
C02599=1072.724,292.709,408.874,174.564,29.541,155.280
C02600=1072.719,292.461,408.906,174.562,29.537,155.279
C02601=1072.713,292.213,408.937,174.558,29.533,155.278
C02602=1072.707,291.965,408.967,174.556,29.529,155.278
C02603=1072.701,291.717,408.997,174.553,29.525,155.277
C02604=1072.694,291.468,409.028,174.550,29.520,155.276
C02605=1072.689,291.221,409.060,174.547,29.516,155.276
C02606=1072.683,290.973,409.090,174.545,29.512,155.275
C02607=1072.678,290.761,409.116,174.542,29.509,155.274
C02608=1072.672,290.548,409.142,174.540,29.505,155.274
C02609=1072.667,290.336,409.168,174.537,29.501,155.273
C02610=1072.662,290.123,409.195,174.534,29.498,155.273
C02611=1072.657,289.911,409.221,174.533,29.494,155.272
C02612=1072.652,289.698,409.247,174.530,29.491,155.271
C02613=1072.647,289.486,409.273,174.528,29.487,155.271
C02614=1072.642,289.274,409.300,174.525,29.484,155.270
C02615=1072.637,289.026,409.330,174.523,29.479,155.269
C02616=1072.630,288.777,409.361,174.520,29.475,155.269
C02617=1072.624,288.529,409.391,174.517,29.471,155.268
C02618=1072.618,288.282,409.421,174.514,29.467,155.267
C02619=1072.612,288.033,409.452,174.512,29.463,155.267
C02620=1072.606,287.785,409.482,174.509,29.459,155.266
C02621=1072.600,287.537,409.513,174.506,29.455,155.265
C02622=1072.594,287.289,409.544,174.503,29.451,155.265
C02623=1072.588,287.041,409.574,174.501,29.447,155.264
C02624=1072.583,286.793,409.604,174.497,29.443,155.263
C02625=1072.576,286.545,409.633,174.495,29.439,155.263
C02626=1072.570,286.297,409.664,174.492,29.435,155.262
C02627=1072.564,286.049,409.694,174.490,29.430,155.261
C02628=1072.558,285.801,409.725,174.486,29.426,155.261
C02629=1072.552,285.553,409.755,174.484,29.422,155.260
C02630=1072.546,285.304,409.785,174.481,29.418,155.259
C02631=1072.540,285.056,409.815,174.479,29.414,155.258
C02632=1072.535,284.808,409.846,174.475,29.410,155.258
C02633=1072.529,284.560,409.876,174.473,29.406,155.257
C02634=1072.523,284.313,409.906,174.470,29.402,155.256
C02635=1072.517,284.063,409.936,174.468,29.398,155.256
C02636=1072.510,283.816,409.966,174.465,29.394,155.255
C02637=1072.504,283.568,409.997,174.462,29.390,155.254
C02638=1072.499,283.320,410.026,174.459,29.386,155.254
C02639=1072.493,283.072,410.057,174.457,29.381,155.253
C02640=1072.487,282.824,410.087,174.454,29.377,155.252
C02641=1072.482,282.576,410.117,174.451,29.373,155.252
C02642=1072.475,282.327,410.147,174.448,29.369,155.251
C02643=1072.469,282.080,410.177,174.446,29.365,155.250
C02644=1072.463,281.831,410.207,174.443,29.361,155.250
C02645=1072.457,281.583,410.237,174.441,29.357,155.249
C02646=1072.452,281.335,410.267,174.437,29.353,155.248
C02647=1072.446,281.087,410.297,174.435,29.349,155.248
C02648=1072.441,280.839,410.327,174.432,29.345,155.247
C02649=1072.434,280.591,410.356,174.430,29.341,155.246
C02650=1072.429,280.343,410.386,174.427,29.337,155.246
C02651=1072.422,280.094,410.417,174.424,29.332,155.245
C02652=1072.417,279.846,410.446,174.421,29.328,155.244
C02653=1072.410,279.598,410.476,174.419,29.324,155.244
C02654=1072.405,279.350,410.506,174.416,29.321,155.243
C02655=1072.398,279.102,410.536,174.414,29.317,155.242
C02656=1072.392,278.854,410.565,174.410,29.312,155.242
C02657=1072.387,278.606,410.595,174.408,29.309,155.241
C02658=1072.380,278.358,410.625,174.405,29.304,155.240
C02659=1072.375,278.109,410.654,174.403,29.300,155.239
C02660=1072.369,277.862,410.685,174.400,29.296,155.239
C02661=1072.363,277.613,410.714,174.398,29.292,155.238
C02662=1072.357,277.365,410.743,174.395,29.288,155.238
C02663=1072.347,276.950,410.793,174.390,29.282,155.236
C02664=1072.337,276.536,410.843,174.386,29.275,155.235
C02665=1072.327,276.121,410.892,174.381,29.268,155.234
C02666=1072.317,275.706,410.941,174.377,29.261,155.233
C02667=1072.312,275.458,410.971,174.374,29.257,155.232
C02668=1072.305,275.210,411.000,174.372,29.254,155.232
C02669=1072.300,274.962,411.030,174.369,29.249,155.231
C02670=1072.294,274.714,411.059,174.367,29.245,155.230
C02671=1072.288,274.465,411.089,174.364,29.241,155.230
C02672=1072.282,274.217,411.118,174.361,29.237,155.229
C02673=1072.276,273.969,411.147,174.359,29.233,155.228
C02674=1072.270,273.721,411.177,174.356,29.229,155.228
C02675=1072.264,273.473,411.207,174.354,29.225,155.227
C02676=1072.258,273.225,411.236,174.351,29.221,155.226
C02677=1072.253,272.976,411.266,174.349,29.218,155.226
C02678=1072.246,272.728,411.295,174.345,29.213,155.225
C02679=1072.241,272.480,411.324,174.343,29.209,155.224
C02680=1072.235,272.232,411.353,174.340,29.205,155.224
C02681=1072.228,271.983,411.382,174.338,29.201,155.223
C02682=1072.223,271.735,411.412,174.335,29.197,155.222
C02683=1072.217,271.487,411.441,174.333,29.193,155.222
C02684=1072.210,271.239,411.470,174.330,29.189,155.221
C02685=1072.205,270.990,411.500,174.327,29.185,155.221
C02686=1072.199,270.743,411.528,174.324,29.181,155.220
C02687=1072.194,270.494,411.558,174.322,29.177,155.219
C02688=1072.187,270.246,411.587,174.319,29.173,155.219
C02689=1072.181,269.998,411.615,174.317,29.169,155.218
C02690=1072.176,269.749,411.645,174.314,29.166,155.217
C02691=1072.170,269.501,411.674,174.312,29.162,155.217
C02692=1072.163,269.253,411.703,174.309,29.158,155.216
C02693=1072.157,269.005,411.732,174.307,29.154,155.215
C02694=1072.152,268.756,411.762,174.303,29.150,155.215
C02695=1072.146,268.509,411.790,174.301,29.146,155.214
C02696=1072.140,268.260,411.819,174.298,29.142,155.213
C02697=1072.134,268.012,411.848,174.296,29.138,155.213
C02698=1072.128,267.763,411.877,174.294,29.134,155.212
C02699=1072.122,267.515,411.906,174.291,29.129,155.211
C02700=1072.116,267.267,411.935,174.289,29.125,155.211
C02701=1072.110,267.018,411.964,174.286,29.121,155.210
C02702=1072.104,266.771,411.992,174.284,29.118,155.209
C02703=1072.099,266.522,412.021,174.281,29.114,155.209
C02704=1072.093,266.274,412.050,174.279,29.110,155.208
C02705=1072.087,266.026,412.079,174.275,29.106,155.207
C02706=1072.081,265.777,412.108,174.273,29.102,155.207
C02707=1072.075,265.530,412.136,174.270,29.098,155.206
C02708=1072.069,265.281,412.166,174.268,29.094,155.206
C02709=1072.063,265.032,412.194,174.265,29.090,155.205
C02710=1072.057,264.784,412.223,174.263,29.086,155.204
C02711=1072.051,264.536,412.252,174.260,29.082,155.204
C02712=1072.046,264.288,412.280,174.258,29.078,155.203
C02713=1072.039,264.040,412.309,174.255,29.074,155.202
C02714=1072.034,263.791,412.338,174.253,29.070,155.202
C02715=1072.024,263.380,412.385,174.249,29.064,155.201
C02716=1072.014,262.969,412.433,174.245,29.057,155.200
C02717=1072.004,262.558,412.480,174.241,29.051,155.198
C02718=1071.994,262.146,412.527,174.235,29.044,155.197
C02719=1071.988,261.898,412.556,174.233,29.040,155.197
C02720=1071.982,261.649,412.584,174.231,29.036,155.196
C02721=1071.976,261.400,412.613,174.228,29.033,155.196
C02722=1071.969,261.152,412.641,174.226,29.029,155.195
C02723=1071.964,260.904,412.669,174.223,29.025,155.194
C02724=1071.957,260.656,412.698,174.221,29.021,155.194
C02725=1071.951,260.407,412.726,174.218,29.017,155.193
C02726=1071.946,260.159,412.755,174.216,29.013,155.192
C02727=1071.940,259.911,412.783,174.213,29.009,155.192
C02728=1071.933,259.663,412.811,174.211,29.005,155.191
C02729=1071.927,259.414,412.840,174.208,29.002,155.191
C02730=1071.922,259.166,412.867,174.206,28.998,155.190
C02731=1071.916,258.918,412.897,174.203,28.994,155.189
C02732=1071.910,258.669,412.925,174.201,28.990,155.189
C02733=1071.904,258.420,412.953,174.198,28.986,155.188
C02734=1071.898,258.173,412.981,174.196,28.982,155.187
C02735=1071.891,257.924,413.010,174.193,28.978,155.187
C02736=1071.886,257.676,413.038,174.191,28.974,155.186
C02737=1071.880,257.428,413.066,174.189,28.970,155.185
C02738=1071.874,257.179,413.094,174.186,28.966,155.185
C02739=1071.868,256.930,413.122,174.184,28.962,155.184
C02740=1071.862,256.682,413.150,174.181,28.958,155.183
C02741=1071.856,256.434,413.179,174.179,28.955,155.183
C02742=1071.851,256.186,413.207,174.176,28.951,155.182
C02743=1071.844,255.938,413.235,174.174,28.947,155.182
C02744=1071.838,255.689,413.263,174.171,28.943,155.181
C02745=1071.833,255.441,413.291,174.169,28.939,155.180
C02746=1071.827,255.192,413.319,174.166,28.935,155.180
C02747=1071.821,254.944,413.347,174.164,28.931,155.179
C02748=1071.815,254.696,413.375,174.161,28.927,155.178
C02749=1071.809,254.447,413.403,174.159,28.923,155.178
C02750=1071.803,254.199,413.431,174.157,28.919,155.177
C02751=1071.797,253.950,413.459,174.154,28.915,155.176
C02752=1071.791,253.702,413.487,174.152,28.911,155.176
C02753=1071.785,253.454,413.515,174.149,28.907,155.175
C02754=1071.780,253.206,413.543,174.147,28.903,155.175
C02755=1071.773,252.957,413.571,174.144,28.899,155.174
C02756=1071.768,252.709,413.599,174.142,28.895,155.173
C02757=1071.762,252.460,413.627,174.139,28.891,155.173
C02758=1071.756,252.212,413.655,174.137,28.888,155.172
C02759=1071.750,251.964,413.683,174.134,28.884,155.171
C02760=1071.744,251.715,413.710,174.132,28.880,155.171
C02761=1071.739,251.466,413.738,174.130,28.876,155.170
C02762=1071.733,251.219,413.766,174.127,28.872,155.169
C02763=1071.727,250.970,413.794,174.125,28.868,155.169
C02764=1071.722,250.722,413.822,174.122,28.864,155.168
C02765=1071.716,250.473,413.850,174.120,28.860,155.167
C02766=1071.710,250.225,413.877,174.117,28.856,155.167
C02767=1071.700,249.811,413.924,174.113,28.849,155.166
C02768=1071.690,249.397,413.970,174.109,28.843,155.165
C02769=1071.681,248.983,414.016,174.105,28.836,155.164
C02770=1071.672,248.570,414.063,174.102,28.830,155.162
C02771=1071.666,248.321,414.090,174.100,28.826,155.162
C02772=1071.660,248.073,414.118,174.097,28.822,155.161
C02773=1071.654,247.824,414.146,174.095,28.818,155.161
C02774=1071.649,247.575,414.173,174.092,28.814,155.160
C02775=1071.643,247.327,414.201,174.090,28.810,155.159
C02776=1071.637,247.079,414.228,174.087,28.806,155.159
C02777=1071.631,246.830,414.256,174.085,28.802,155.158
C02778=1071.625,246.582,414.283,174.083,28.798,155.157
C02779=1071.619,246.334,414.311,174.080,28.794,155.157
C02780=1071.614,246.085,414.338,174.078,28.790,155.156
C02781=1071.608,245.837,414.366,174.075,28.786,155.155
C02782=1071.602,245.588,414.393,174.073,28.782,155.155
C02783=1071.596,245.340,414.421,174.070,28.778,155.154
C02784=1071.590,245.091,414.448,174.069,28.774,155.153
C02785=1071.585,244.843,414.476,174.066,28.770,155.153
C02786=1071.579,244.594,414.503,174.064,28.766,155.152
C02787=1071.572,244.346,414.530,174.062,28.762,155.151
C02788=1071.567,244.098,414.558,174.059,28.758,155.151
C02789=1071.561,243.849,414.585,174.057,28.755,155.150
C02790=1071.556,243.601,414.613,174.054,28.751,155.150
C02791=1071.550,243.352,414.639,174.052,28.747,155.149
C02792=1071.543,243.104,414.667,174.049,28.743,155.148
C02793=1071.538,242.855,414.694,174.047,28.739,155.148
C02794=1071.532,242.607,414.722,174.045,28.735,155.147
C02795=1071.526,242.358,414.749,174.043,28.731,155.146
C02796=1071.521,242.110,414.776,174.041,28.727,155.146
C02797=1071.515,241.862,414.803,174.038,28.723,155.145
C02798=1071.508,241.613,414.830,174.036,28.719,155.145
C02799=1071.503,241.364,414.857,174.033,28.715,155.144
C02800=1071.497,241.116,414.885,174.031,28.711,155.143
C02801=1071.491,240.867,414.912,174.029,28.707,155.143
C02802=1071.485,240.619,414.938,174.026,28.704,155.142
C02803=1071.479,240.371,414.965,174.024,28.700,155.141
C02804=1071.473,240.122,414.993,174.022,28.696,155.141
C02805=1071.468,239.873,415.020,174.020,28.692,155.140
C02806=1071.462,239.625,415.047,174.017,28.688,155.139
C02807=1071.455,239.376,415.074,174.015,28.684,155.139
C02808=1071.449,239.128,415.101,174.012,28.680,155.138
C02809=1071.444,238.880,415.128,174.010,28.676,155.138
C02810=1071.438,238.632,415.154,174.008,28.672,155.137
C02811=1071.431,238.383,415.181,174.005,28.668,155.136
C02812=1071.426,238.134,415.209,174.004,28.665,155.136
C02813=1071.421,237.886,415.235,174.001,28.661,155.135
C02814=1071.415,237.637,415.262,173.999,28.657,155.134
C02815=1071.408,237.389,415.290,173.996,28.653,155.134
C02816=1071.402,237.140,415.316,173.994,28.649,155.133
C02817=1071.397,236.892,415.343,173.992,28.645,155.133
C02818=1071.391,236.644,415.370,173.989,28.641,155.132
C02819=1071.381,236.222,415.415,173.986,28.634,155.131
C02820=1071.371,235.802,415.460,173.982,28.628,155.130
C02821=1071.361,235.382,415.506,173.978,28.621,155.129
C02822=1071.352,234.961,415.551,173.974,28.614,155.128
C02823=1071.346,234.713,415.577,173.972,28.610,155.127
C02824=1071.340,234.464,415.604,173.969,28.606,155.126
C02825=1071.334,234.216,415.631,173.968,28.603,155.126
C02826=1071.328,233.967,415.658,173.965,28.599,155.125
C02827=1071.322,233.719,415.684,173.963,28.595,155.124
C02828=1071.317,233.471,415.711,173.961,28.591,155.124
C02829=1071.311,233.222,415.738,173.958,28.587,155.123
C02830=1071.304,232.973,415.765,173.956,28.583,155.122
C02831=1071.299,232.725,415.791,173.954,28.579,155.122
C02832=1071.293,232.476,415.818,173.952,28.575,155.121
C02833=1071.287,232.228,415.844,173.949,28.571,155.120
C02834=1071.282,231.979,415.870,173.947,28.567,155.120
C02835=1071.276,231.731,415.897,173.945,28.563,155.119
C02836=1071.270,231.482,415.924,173.942,28.559,155.119
C02837=1071.264,231.234,415.950,173.941,28.555,155.118
C02838=1071.258,230.984,415.977,173.938,28.551,155.117
C02839=1071.252,230.736,416.003,173.936,28.547,155.117
C02840=1071.246,230.488,416.029,173.934,28.543,155.116
C02841=1071.240,230.240,416.056,173.931,28.540,155.115
C02842=1071.235,229.991,416.082,173.930,28.536,155.115
C02843=1071.229,229.742,416.109,173.927,28.532,155.114
C02844=1071.223,229.494,416.135,173.925,28.528,155.114
C02845=1071.218,229.245,416.161,173.922,28.524,155.113
C02846=1071.211,228.997,416.187,173.920,28.520,155.112
C02847=1071.205,228.748,416.214,173.919,28.516,155.112
C02848=1071.199,228.499,416.240,173.916,28.512,155.111
C02849=1071.194,228.250,416.267,173.914,28.508,155.110
C02850=1071.187,228.002,416.293,173.911,28.504,155.110
C02851=1071.182,227.753,416.319,173.909,28.500,155.109
C02852=1071.176,227.505,416.345,173.908,28.497,155.108
C02853=1071.170,227.256,416.371,173.905,28.493,155.108
C02854=1071.164,227.008,416.397,173.903,28.489,155.107
C02855=1071.158,226.760,416.424,173.900,28.485,155.107
C02856=1071.153,226.511,416.450,173.898,28.481,155.106
C02857=1071.146,226.263,416.476,173.897,28.477,155.105
C02858=1071.141,226.014,416.502,173.894,28.473,155.105
C02859=1071.135,225.765,416.529,173.892,28.469,155.104
C02860=1071.129,225.517,416.554,173.889,28.465,155.103
C02861=1071.123,225.268,416.581,173.888,28.461,155.103
C02862=1071.117,225.019,416.607,173.886,28.457,155.102
C02863=1071.111,224.771,416.633,173.883,28.453,155.101
C02864=1071.105,224.522,416.659,173.881,28.449,155.101
C02865=1071.100,224.273,416.685,173.878,28.445,155.100
C02866=1071.093,224.025,416.711,173.877,28.441,155.099
C02867=1071.088,223.776,416.736,173.875,28.437,155.099
C02868=1071.082,223.528,416.763,173.872,28.433,155.098
C02869=1071.076,223.279,416.788,173.870,28.429,155.098
C02870=1071.071,223.030,416.814,173.868,28.425,155.097
C02871=1071.065,222.816,416.837,173.866,28.422,155.096
C02872=1071.061,222.602,416.860,173.864,28.419,155.096
C02873=1071.056,222.388,416.882,173.863,28.416,155.095
C02874=1071.050,222.173,416.904,173.860,28.412,155.095
C02875=1071.045,221.960,416.926,173.859,28.408,155.094
C02876=1071.041,221.745,416.949,173.857,28.405,155.094
C02877=1071.035,221.531,416.971,173.855,28.402,155.093
C02878=1071.030,221.316,416.994,173.854,28.398,155.092
C02879=1071.024,221.067,417.019,173.851,28.394,155.092
C02880=1071.018,220.818,417.045,173.849,28.390,155.091
C02881=1071.013,220.571,417.071,173.846,28.386,155.091
C02882=1071.007,220.322,417.097,173.845,28.382,155.090
C02883=1071.001,220.073,417.122,173.843,28.378,155.089
C02884=1070.995,219.824,417.148,173.840,28.374,155.089
C02885=1070.989,219.576,417.174,173.838,28.370,155.088
C02886=1070.983,219.328,417.199,173.836,28.367,155.087
C02887=1070.977,219.079,417.225,173.834,28.363,155.087
C02888=1070.971,218.830,417.250,173.832,28.359,155.086
C02889=1070.966,218.581,417.276,173.830,28.355,155.086
C02890=1070.959,218.332,417.302,173.828,28.351,155.085
C02891=1070.953,218.084,417.327,173.825,28.347,155.084
C02892=1070.948,217.836,417.353,173.823,28.343,155.084
C02893=1070.942,217.587,417.379,173.822,28.339,155.083
C02894=1070.936,217.338,417.405,173.819,28.335,155.082
C02895=1070.930,217.090,417.430,173.817,28.331,155.082
C02896=1070.924,216.841,417.455,173.814,28.327,155.081
C02897=1070.918,216.592,417.481,173.813,28.324,155.080
C02898=1070.912,216.343,417.507,173.811,28.319,155.080
C02899=1070.907,216.095,417.532,173.808,28.315,155.079
C02900=1070.901,215.847,417.557,173.807,28.312,155.078
C02901=1070.895,215.598,417.583,173.805,28.308,155.078
C02902=1070.889,215.349,417.609,173.802,28.304,155.077
C02903=1070.883,215.100,417.634,173.801,28.300,155.077
C02904=1070.878,214.852,417.659,173.798,28.296,155.076
C02905=1070.872,214.603,417.685,173.796,28.291,155.075
C02906=1070.866,214.355,417.710,173.794,28.287,155.074
C02907=1070.860,214.106,417.736,173.792,28.283,155.074
C02908=1070.855,213.858,417.761,173.790,28.279,155.073
C02909=1070.849,213.609,417.787,173.788,28.275,155.073
C02910=1070.842,213.360,417.812,173.786,28.271,155.072
C02911=1070.837,213.111,417.838,173.784,28.267,155.071
C02912=1070.832,212.863,417.862,173.781,28.263,155.071
C02913=1070.825,212.614,417.887,173.780,28.260,155.070
C02914=1070.819,212.365,417.913,173.778,28.256,155.069
C02915=1070.814,212.116,417.939,173.775,28.251,155.069
C02916=1070.808,211.868,417.964,173.774,28.248,155.068
C02917=1070.802,211.620,417.989,173.772,28.244,155.067
C02918=1070.796,211.370,418.014,173.769,28.240,155.067
C02919=1070.790,211.122,418.039,173.768,28.236,155.066
C02920=1070.784,210.874,418.064,173.765,28.232,155.065
C02921=1070.779,210.625,418.090,173.763,28.228,155.065
C02922=1070.773,210.376,418.114,173.761,28.224,155.064
C02923=1070.767,210.127,418.140,173.759,28.220,155.064
C02924=1070.761,209.879,418.165,173.757,28.216,155.063
C02925=1070.755,209.630,418.190,173.755,28.212,155.062
C02926=1070.749,209.381,418.215,173.753,28.208,155.062
C02927=1070.744,209.170,418.236,173.752,28.205,155.061
C02928=1070.739,208.958,418.258,173.749,28.201,155.060
C02929=1070.734,208.745,418.279,173.748,28.197,155.060
C02930=1070.729,208.533,418.300,173.746,28.194,155.059
C02931=1070.725,208.321,418.322,173.744,28.191,155.059
C02932=1070.719,208.109,418.343,173.742,28.187,155.058
C02933=1070.714,207.897,418.364,173.741,28.184,155.058
C02934=1070.685,206.642,418.488,173.603,28.111,155.055
C02935=1070.680,206.393,418.512,173.601,28.108,155.054
C02936=1070.674,206.145,418.536,173.599,28.104,155.054
C02937=1070.668,205.896,418.560,173.596,28.101,155.054
C02938=1070.662,205.648,418.585,173.594,28.098,155.053
C02939=1070.657,205.399,418.609,173.592,28.095,155.053
C02940=1070.650,205.150,418.633,173.590,28.092,155.052
C02941=1070.645,204.901,418.657,173.587,28.089,155.052
C02942=1070.640,204.652,418.681,173.586,28.086,155.051
C02943=1070.634,204.403,418.706,173.583,28.083,155.051
C02944=1070.628,204.155,418.729,173.581,28.080,155.051
C02945=1070.623,203.906,418.754,173.578,28.077,155.050
C02946=1070.617,203.657,418.778,173.577,28.074,155.050
C02947=1070.612,203.408,418.803,173.574,28.071,155.049
C02948=1070.606,203.160,418.826,173.572,28.068,155.049
C02949=1070.600,202.911,418.851,173.570,28.064,155.048
C02950=1070.594,202.662,418.875,173.568,28.061,155.048
C02951=1070.589,202.413,418.899,173.565,28.059,155.048
C02952=1070.583,202.165,418.923,173.564,28.056,155.047
C02953=1070.577,201.915,418.947,173.561,28.052,155.047
C02954=1070.571,201.667,418.971,173.559,28.049,155.046
C02955=1070.566,201.418,418.995,173.556,28.046,155.046
C02956=1070.560,201.169,419.019,173.555,28.044,155.045
C02957=1070.554,200.921,419.043,173.552,28.041,155.045
C02958=1070.548,200.672,419.066,173.550,28.038,155.045
C02959=1070.542,200.423,419.090,173.548,28.035,155.044
C02960=1070.537,200.174,419.114,173.546,28.032,155.044
C02961=1070.531,199.926,419.138,173.543,28.028,155.043
C02962=1070.525,199.676,419.162,173.542,28.026,155.043
C02963=1070.519,199.428,419.186,173.539,28.023,155.043
C02964=1070.514,199.179,419.210,173.537,28.020,155.042
C02965=1070.508,198.930,419.233,173.535,28.017,155.042
C02966=1070.502,198.681,419.257,173.533,28.014,155.041
C02967=1070.496,198.433,419.281,173.530,28.011,155.041
C02968=1070.491,198.184,419.305,173.529,28.008,155.040
C02969=1070.485,197.935,419.328,173.526,28.005,155.040
C02970=1070.478,197.686,419.352,173.524,28.002,155.040
C02971=1070.473,197.437,419.376,173.522,27.999,155.039
C02972=1070.467,197.189,419.400,173.520,27.996,155.039
C02973=1070.462,196.940,419.424,173.517,27.993,155.038
C02974=1070.456,196.691,419.447,173.516,27.990,155.038
C02975=1070.450,196.442,419.471,173.513,27.987,155.038
C02976=1070.445,196.193,419.494,173.511,27.984,155.037
C02977=1070.439,195.945,419.518,173.509,27.981,155.037
C02978=1070.433,195.696,419.542,173.507,27.978,155.036
C02979=1070.427,195.447,419.566,173.504,27.975,155.036
C02980=1070.422,195.198,419.590,173.503,27.972,155.036
C02981=1070.416,194.949,419.613,173.500,27.969,155.035
C02982=1070.410,194.701,419.636,173.499,27.967,155.035
C02983=1070.405,194.452,419.660,173.496,27.964,155.034
C02984=1070.399,194.204,419.684,173.494,27.960,155.034
C02985=1070.392,193.954,419.707,173.492,27.957,155.033
C02986=1070.387,193.705,419.731,173.490,27.955,155.033
C02987=1070.381,193.456,419.754,173.487,27.952,155.033
C02988=1070.376,193.208,419.778,173.486,27.949,155.032
C02989=1070.370,192.959,419.801,173.483,27.946,155.032
C02990=1070.365,192.710,419.824,173.482,27.943,155.031
C02991=1070.359,192.462,419.849,173.479,27.940,155.031
C02992=1070.354,192.213,419.871,173.477,27.937,155.031
C02993=1070.347,191.964,419.896,173.475,27.934,155.030
C02994=1070.342,191.714,419.919,173.473,27.931,155.030
C02995=1070.336,191.433,419.945,173.470,27.927,155.029
C02996=1070.329,191.151,419.972,173.468,27.924,155.029
C02997=1070.323,190.869,419.998,173.465,27.921,155.028
C02998=1070.316,190.587,420.025,173.463,27.917,155.028
C02999=1070.310,190.338,420.049,173.461,27.914,155.027
C03000=1070.305,190.089,420.072,173.459,27.911,155.027
C03001=1070.299,189.840,420.095,173.457,27.909,155.027
C03002=1070.294,189.591,420.118,173.455,27.906,155.026
C03003=1070.288,189.343,420.142,173.453,27.903,155.026
C03004=1070.283,189.094,420.165,173.451,27.900,155.025
C03005=1070.277,188.845,420.188,173.448,27.896,155.025
C03006=1070.272,188.596,420.212,173.447,27.894,155.025
C03007=1070.266,188.347,420.235,173.444,27.891,155.024
C03008=1070.260,188.099,420.258,173.443,27.888,155.024
C03009=1070.255,187.849,420.282,173.440,27.885,155.023
C03010=1070.249,187.600,420.305,173.439,27.882,155.023
C03011=1070.243,187.352,420.328,173.436,27.879,155.023
C03012=1070.238,187.103,420.351,173.434,27.876,155.022
C03013=1070.233,186.854,420.375,173.432,27.873,155.022
C03014=1070.227,186.605,420.398,173.430,27.870,155.021
C03015=1070.221,186.356,420.421,173.428,27.867,155.021
C03016=1070.216,186.107,420.444,173.426,27.864,155.020
C03017=1070.210,185.859,420.468,173.424,27.862,155.020
C03018=1070.204,185.610,420.491,173.422,27.859,155.020
C03019=1070.199,185.361,420.514,173.420,27.855,155.019
C03020=1070.194,185.113,420.537,173.418,27.852,155.019
C03021=1070.189,184.864,420.560,173.416,27.850,155.018
C03022=1070.183,184.615,420.583,173.414,27.847,155.018
C03023=1070.177,184.365,420.606,173.411,27.844,155.018
C03024=1070.171,184.116,420.629,173.410,27.841,155.017
C03025=1070.164,183.868,420.652,173.407,27.838,155.017
C03026=1070.159,183.619,420.675,173.406,27.836,155.017
C03027=1070.153,183.370,420.698,173.403,27.833,155.016
C03028=1070.147,183.121,420.720,173.402,27.830,155.016
C03029=1070.141,182.872,420.743,173.399,27.827,155.015
C03030=1070.136,182.623,420.766,173.398,27.824,155.015
C03031=1070.129,182.375,420.789,173.395,27.821,155.015
C03032=1070.124,182.126,420.812,173.394,27.818,155.014
C03033=1070.118,181.877,420.835,173.391,27.815,155.014
C03034=1070.112,181.628,420.858,173.389,27.813,155.013
C03035=1070.106,181.379,420.880,173.387,27.810,155.013
C03036=1070.101,181.130,420.903,173.385,27.807,155.013
C03037=1070.094,180.882,420.926,173.383,27.804,155.012
C03038=1070.089,180.632,420.948,173.381,27.801,155.012
C03039=1070.083,180.383,420.971,173.379,27.799,155.011
C03040=1070.077,180.134,420.994,173.377,27.796,155.011
C03041=1070.072,179.885,421.017,173.375,27.793,155.011
C03042=1070.065,179.637,421.039,173.373,27.790,155.010
C03043=1070.059,179.388,421.062,173.371,27.788,155.010
C03044=1070.054,179.139,421.085,173.368,27.785,155.010
C03045=1070.048,178.889,421.107,173.367,27.782,155.009
C03046=1070.043,178.641,421.130,173.364,27.779,155.009
C03047=1070.037,178.393,421.152,173.363,27.776,155.008
C03048=1070.031,178.144,421.175,173.360,27.773,155.008
C03049=1070.025,177.895,421.198,173.359,27.771,155.008
C03050=1070.020,177.645,421.220,173.356,27.768,155.007
C03051=1070.013,177.397,421.243,173.355,27.765,155.007
C03052=1070.007,177.148,421.266,173.352,27.762,155.006
C03053=1070.002,176.898,421.288,173.351,27.759,155.006
C03054=1069.996,176.649,421.311,173.348,27.757,155.006
C03055=1069.990,176.401,421.333,173.347,27.754,155.005
C03056=1069.985,176.153,421.356,173.344,27.751,155.005
C03057=1069.979,175.903,421.378,173.343,27.748,155.005
C03058=1069.974,175.654,421.401,173.340,27.745,155.004
C03059=1069.967,175.372,421.426,173.339,27.742,155.004
C03060=1069.960,175.089,421.452,173.336,27.739,155.003
C03061=1069.953,174.807,421.477,173.334,27.736,155.003
C03062=1069.948,174.525,421.503,173.332,27.732,155.002
C03063=1069.941,174.276,421.525,173.330,27.729,155.002
C03064=1069.935,174.027,421.548,173.328,27.726,155.002
C03065=1069.930,173.778,421.570,173.326,27.724,155.001
C03066=1069.925,173.529,421.593,173.324,27.721,155.001
C03067=1069.919,173.280,421.615,173.322,27.718,155.001
C03068=1069.913,173.031,421.637,173.320,27.716,155.000
C03069=1069.907,172.782,421.660,173.318,27.713,155.000
C03070=1069.902,172.534,421.682,173.316,27.710,154.999
C03071=1069.896,172.285,421.705,173.314,27.707,154.999
C03072=1069.890,172.035,421.727,173.312,27.704,154.999
C03073=1069.885,171.787,421.750,173.310,27.701,154.998
C03074=1069.879,171.538,421.771,173.308,27.698,154.998
C03075=1069.873,171.289,421.794,173.306,27.695,154.997
C03076=1069.868,171.040,421.816,173.304,27.693,154.997
C03077=1069.861,170.791,421.839,173.303,27.690,154.997
C03078=1069.857,170.542,421.860,173.300,27.687,154.996
C03079=1069.851,170.293,421.883,173.299,27.684,154.996
C03080=1069.845,170.044,421.905,173.296,27.681,154.995
C03081=1069.839,169.795,421.928,173.295,27.678,154.995
C03082=1069.834,169.546,421.950,173.292,27.675,154.995
C03083=1069.828,169.297,421.971,173.291,27.673,154.994
C03084=1069.822,169.048,421.994,173.289,27.670,154.994
C03085=1069.817,168.799,422.017,173.287,27.667,154.993
C03086=1069.811,168.551,422.039,173.285,27.664,154.993
C03087=1069.806,168.301,422.061,173.283,27.662,154.993
C03088=1069.800,168.052,422.083,173.281,27.659,154.992
C03089=1069.794,167.804,422.105,173.279,27.656,154.992
C03090=1069.789,167.554,422.127,173.277,27.653,154.991
C03091=1069.783,167.306,422.150,173.276,27.650,154.991
C03092=1069.778,167.057,422.172,173.273,27.647,154.991
C03093=1069.772,166.808,422.194,173.272,27.645,154.990
C03094=1069.766,166.559,422.216,173.269,27.642,154.990
C03095=1069.761,166.310,422.238,173.268,27.639,154.990
C03096=1069.755,166.061,422.260,173.266,27.636,154.989
C03097=1069.750,165.812,422.281,173.264,27.633,154.989
C03098=1069.744,165.563,422.304,173.262,27.630,154.988
C03099=1069.739,165.314,422.327,173.261,27.627,154.988
C03100=1069.733,165.065,422.348,173.258,27.624,154.988
C03101=1069.728,164.816,422.370,173.257,27.622,154.987
C03102=1069.721,164.567,422.393,173.254,27.619,154.987
C03103=1069.716,164.318,422.414,173.253,27.616,154.986
C03104=1069.711,164.069,422.437,173.251,27.613,154.986
C03105=1069.705,163.820,422.458,173.249,27.610,154.986
C03106=1069.700,163.571,422.481,173.247,27.607,154.985
C03107=1069.694,163.323,422.502,173.245,27.604,154.985
C03108=1069.689,163.073,422.524,173.243,27.602,154.984
C03109=1069.683,162.824,422.547,173.242,27.599,154.984
C03110=1069.678,162.575,422.568,173.239,27.596,154.984
C03111=1069.672,162.326,422.590,173.238,27.593,154.983
C03112=1069.666,162.078,422.612,173.236,27.590,154.983
C03113=1069.661,161.828,422.634,173.234,27.587,154.982
C03114=1069.655,161.580,422.656,173.232,27.584,154.982
C03115=1069.650,161.330,422.678,173.231,27.582,154.982
C03116=1069.644,161.081,422.699,173.229,27.579,154.981
C03117=1069.639,160.832,422.721,173.227,27.576,154.981
C03118=1069.633,160.583,422.743,173.225,27.573,154.980
C03119=1069.627,160.335,422.764,173.223,27.570,154.980
C03120=1069.621,160.085,422.786,173.222,27.567,154.980
C03121=1069.616,159.836,422.808,173.219,27.565,154.979
C03122=1069.610,159.587,422.829,173.217,27.562,154.979
C03123=1069.603,159.305,422.854,173.215,27.559,154.978
C03124=1069.597,159.023,422.879,173.214,27.556,154.978
C03125=1069.590,158.739,422.903,173.211,27.553,154.978
C03126=1069.584,158.457,422.928,173.209,27.549,154.977
C03127=1069.578,158.208,422.949,173.207,27.546,154.977
C03128=1069.573,157.958,422.971,173.206,27.544,154.976
C03129=1069.567,157.710,422.993,173.203,27.541,154.976
C03130=1069.561,157.461,423.014,173.202,27.538,154.976
C03131=1069.555,157.212,423.035,173.200,27.536,154.975
C03132=1069.550,156.963,423.058,173.198,27.533,154.975
C03133=1069.544,156.714,423.079,173.196,27.530,154.974
C03134=1069.538,156.465,423.101,173.195,27.527,154.974
C03135=1069.532,156.216,423.122,173.192,27.525,154.974
C03136=1069.527,155.967,423.143,173.191,27.522,154.973
C03137=1069.521,155.717,423.165,173.189,27.519,154.973
C03138=1069.516,155.469,423.186,173.187,27.516,154.973
C03139=1069.510,155.219,423.208,173.185,27.513,154.972
C03140=1069.504,154.971,423.229,173.184,27.510,154.972
C03141=1069.498,154.722,423.251,173.181,27.508,154.971
C03142=1069.492,154.473,423.272,173.180,27.505,154.971
C03143=1069.486,154.223,423.293,173.178,27.502,154.971
C03144=1069.482,153.975,423.315,173.176,27.499,154.970
C03145=1069.475,153.725,423.337,173.174,27.497,154.970
C03146=1069.470,153.477,423.358,173.173,27.494,154.969
C03147=1069.464,153.227,423.379,173.170,27.491,154.969
C03148=1069.458,152.979,423.400,173.169,27.489,154.969
C03149=1069.452,152.729,423.422,173.167,27.486,154.968
C03150=1069.447,152.481,423.443,173.165,27.483,154.968
C03151=1069.441,152.231,423.464,173.163,27.480,154.968
C03152=1069.435,151.983,423.485,173.162,27.477,154.967
C03153=1069.429,151.733,423.507,173.159,27.475,154.967
C03154=1069.424,151.485,423.528,173.158,27.472,154.967
C03155=1069.418,151.235,423.549,173.156,27.469,154.966
C03156=1069.412,150.987,423.570,173.155,27.467,154.966
C03157=1069.406,150.737,423.592,173.152,27.463,154.965
C03158=1069.402,150.488,423.613,173.151,27.461,154.965
C03159=1069.396,150.239,423.634,173.149,27.458,154.965
C03160=1069.390,149.990,423.656,173.147,27.455,154.964
C03161=1069.385,149.741,423.676,173.145,27.453,154.964
C03162=1069.378,149.492,423.698,173.144,27.450,154.963
C03163=1069.373,149.243,423.719,173.142,27.447,154.963
C03164=1069.367,148.994,423.740,173.140,27.444,154.963
C03165=1069.361,148.745,423.761,173.138,27.441,154.962
C03166=1069.356,148.496,423.782,173.137,27.439,154.962
C03167=1069.349,148.247,423.803,173.134,27.436,154.962
C03168=1069.344,147.998,423.824,173.133,27.433,154.961
C03169=1069.338,147.749,423.845,173.131,27.431,154.961
C03170=1069.332,147.500,423.867,173.130,27.428,154.960
C03171=1069.326,147.250,423.887,173.127,27.425,154.960
C03172=1069.321,147.002,423.909,173.126,27.422,154.960
C03173=1069.316,146.753,423.929,173.124,27.420,154.959
C03174=1069.309,146.503,423.951,173.122,27.417,154.959
C03175=1069.303,146.255,423.971,173.120,27.414,154.958
C03176=1069.297,146.005,423.993,173.119,27.412,154.958
C03177=1069.292,145.756,424.013,173.117,27.409,154.958
C03178=1069.286,145.508,424.034,173.115,27.406,154.957
C03179=1069.281,145.258,424.055,173.113,27.403,154.957
C03180=1069.275,145.010,424.077,173.112,27.400,154.957
C03181=1069.268,144.760,424.097,173.110,27.398,154.956
C03182=1069.263,144.512,424.118,173.108,27.395,154.956
C03183=1069.258,144.262,424.139,173.106,27.392,154.956
C03184=1069.252,144.013,424.160,173.105,27.389,154.955
C03185=1069.246,143.764,424.181,173.102,27.386,154.955
C03186=1069.240,143.515,424.201,173.101,27.384,154.954
C03187=1069.234,143.233,424.225,173.099,27.381,154.954
C03188=1069.228,142.949,424.249,173.097,27.378,154.954
C03189=1069.221,142.666,424.272,173.095,27.374,154.953
C03190=1069.214,142.383,424.296,173.093,27.371,154.953
C03191=1069.209,142.134,424.317,173.091,27.369,154.952
C03192=1069.203,141.884,424.338,173.090,27.366,154.952
C03193=1069.197,141.636,424.358,173.087,27.363,154.952
C03194=1069.192,141.387,424.379,173.086,27.361,154.951
C03195=1069.186,141.137,424.400,173.084,27.358,154.951
C03196=1069.180,140.889,424.421,173.083,27.355,154.950
C03197=1069.174,140.640,424.441,173.080,27.352,154.950
C03198=1069.168,140.390,424.462,173.079,27.349,154.950
C03199=1069.163,140.142,424.483,173.077,27.347,154.949
C03200=1069.158,139.893,424.504,173.076,27.344,154.949
C03201=1069.151,139.643,424.524,173.073,27.341,154.949
C03202=1069.146,139.394,424.545,173.072,27.338,154.948
C03203=1069.141,139.145,424.565,173.071,27.336,154.948
C03204=1069.134,138.897,424.586,173.069,27.333,154.947
C03205=1069.128,138.647,424.607,173.066,27.330,154.947
C03206=1069.122,138.398,424.627,173.065,27.328,154.947
C03207=1069.117,138.149,424.647,173.064,27.325,154.946
C03208=1069.111,137.900,424.669,173.062,27.322,154.946
C03209=1069.105,137.651,424.689,173.060,27.320,154.946
C03210=1069.100,137.402,424.709,173.058,27.317,154.945
C03211=1069.094,137.153,424.729,173.057,27.314,154.945
C03212=1069.088,136.903,424.750,173.055,27.311,154.944
C03213=1069.083,136.654,424.771,173.054,27.308,154.944
C03214=1069.077,136.405,424.791,173.051,27.306,154.944
C03215=1069.071,136.157,424.812,173.050,27.303,154.943
C03216=1069.064,135.907,424.832,173.048,27.300,154.943
C03217=1069.059,135.658,424.853,173.047,27.297,154.942
C03218=1069.053,135.409,424.873,173.045,27.295,154.942
C03219=1069.048,135.160,424.894,173.043,27.292,154.942
C03220=1069.042,134.910,424.914,173.041,27.289,154.941
C03221=1069.036,134.661,424.934,173.040,27.287,154.941
C03222=1069.031,134.412,424.955,173.038,27.284,154.941
C03223=1069.025,134.163,424.975,173.037,27.281,154.940
C03224=1069.019,133.914,424.996,173.034,27.279,154.940
C03225=1069.013,133.665,425.016,173.033,27.276,154.940
C03226=1069.008,133.416,425.036,173.031,27.273,154.939
C03227=1069.002,133.167,425.056,173.030,27.270,154.939
C03228=1068.996,132.918,425.077,173.028,27.267,154.938
C03229=1068.990,132.669,425.097,173.026,27.264,154.938
C03230=1068.985,132.419,425.118,173.024,27.262,154.938
C03231=1068.979,132.170,425.138,173.023,27.259,154.937
C03232=1068.973,131.921,425.158,173.021,27.257,154.937
C03233=1068.967,131.672,425.178,173.020,27.254,154.936
C03234=1068.962,131.423,425.199,173.017,27.251,154.936
C03235=1068.956,131.174,425.219,173.016,27.248,154.936
C03236=1068.950,130.925,425.239,173.014,27.246,154.935
C03237=1068.944,130.676,425.259,173.013,27.243,154.935
C03238=1068.938,130.427,425.280,173.011,27.241,154.935
C03239=1068.932,130.177,425.300,173.009,27.238,154.934
C03240=1068.926,129.929,425.320,173.007,27.235,154.934
C03241=1068.921,129.679,425.340,173.006,27.233,154.934
C03242=1068.915,129.430,425.360,173.004,27.230,154.933
C03243=1068.909,129.181,425.380,173.003,27.227,154.933
C03244=1068.902,128.932,425.400,173.000,27.224,154.932
C03245=1068.897,128.683,425.420,172.999,27.222,154.932
C03246=1068.891,128.434,425.440,172.997,27.219,154.932
C03247=1068.885,128.184,425.460,172.996,27.216,154.931
C03248=1068.879,127.936,425.480,172.994,27.213,154.931
C03249=1068.874,127.686,425.500,172.993,27.211,154.931
C03250=1068.867,127.437,425.521,172.990,27.208,154.930
C03251=1068.861,127.155,425.543,172.989,27.205,154.930
C03252=1068.855,126.871,425.566,172.986,27.202,154.929
C03253=1068.848,126.588,425.589,172.985,27.199,154.929
C03254=1068.841,126.304,425.611,172.983,27.196,154.929
C03255=1068.835,126.056,425.631,172.981,27.193,154.928
C03256=1068.829,125.807,425.651,172.980,27.190,154.928
C03257=1068.824,125.558,425.671,172.978,27.188,154.927
C03258=1068.818,125.308,425.691,172.977,27.185,154.927
C03259=1068.812,125.059,425.711,172.975,27.182,154.927
C03260=1068.806,124.811,425.731,172.974,27.179,154.926
C03261=1068.800,124.562,425.750,172.971,27.176,154.926
C03262=1068.795,124.311,425.771,172.970,27.174,154.926
C03263=1068.789,124.062,425.791,172.968,27.171,154.925
C03264=1068.783,123.814,425.811,172.967,27.169,154.925
C03265=1068.777,123.564,425.830,172.965,27.166,154.924
C03266=1068.772,123.315,425.850,172.964,27.163,154.924
C03267=1068.766,123.066,425.870,172.961,27.160,154.924
C03268=1068.760,122.817,425.890,172.960,27.158,154.923
C03269=1068.754,122.568,425.910,172.958,27.155,154.923
C03270=1068.748,122.319,425.929,172.957,27.152,154.923
C03271=1068.742,122.070,425.949,172.955,27.149,154.922
C03272=1068.737,121.821,425.969,172.954,27.147,154.922
C03273=1068.731,121.571,425.989,172.952,27.144,154.921
C03274=1068.725,121.322,426.009,172.950,27.141,154.921
C03275=1068.720,121.073,426.028,172.948,27.138,154.921
C03276=1068.714,120.824,426.048,172.947,27.136,154.920
C03277=1068.709,120.574,426.068,172.945,27.133,154.920
C03278=1068.703,120.326,426.088,172.944,27.131,154.920
C03279=1068.697,120.077,426.107,172.942,27.128,154.919
C03280=1068.691,119.827,426.127,172.941,27.125,154.919
C03281=1068.685,119.579,426.147,172.939,27.122,154.918
C03282=1068.680,119.329,426.166,172.937,27.119,154.918
C03283=1068.674,119.080,426.186,172.936,27.116,154.918
C03284=1068.669,118.831,426.206,172.934,27.114,154.917
C03285=1068.663,118.582,426.226,172.932,27.111,154.917
C03286=1068.657,118.332,426.245,172.931,27.108,154.916
C03287=1068.651,118.083,426.264,172.930,27.106,154.916
C03288=1068.645,117.834,426.284,172.928,27.103,154.916
C03289=1068.640,117.585,426.303,172.926,27.100,154.915
C03290=1068.634,117.336,426.324,172.924,27.097,154.915
C03291=1068.629,117.086,426.343,172.923,27.095,154.915
C03292=1068.623,116.837,426.363,172.921,27.092,154.914
C03293=1068.617,116.588,426.382,172.920,27.089,154.914
C03294=1068.611,116.339,426.402,172.918,27.086,154.913
C03295=1068.605,116.090,426.422,172.917,27.084,154.913
C03296=1068.600,115.840,426.441,172.915,27.081,154.913
C03297=1068.594,115.592,426.460,172.914,27.078,154.912
C03298=1068.589,115.342,426.480,172.911,27.075,154.912
C03299=1068.583,115.093,426.500,172.910,27.072,154.911
C03300=1068.577,114.844,426.519,172.908,27.070,154.911
C03301=1068.572,114.595,426.539,172.907,27.067,154.911
C03302=1068.566,114.345,426.558,172.905,27.064,154.910
C03303=1068.560,114.096,426.578,172.904,27.061,154.910
C03304=1068.554,113.847,426.597,172.903,27.059,154.909
C03305=1068.549,113.598,426.616,172.901,27.056,154.909
C03306=1068.543,113.349,426.636,172.899,27.054,154.909
C03307=1068.537,113.099,426.656,172.897,27.050,154.908
C03308=1068.531,112.850,426.675,172.896,27.048,154.908
C03309=1068.526,112.601,426.693,172.894,27.045,154.908
C03310=1068.520,112.353,426.713,172.893,27.042,154.907
C03311=1068.514,112.103,426.732,172.891,27.040,154.907
C03312=1068.508,111.854,426.752,172.890,27.037,154.907
C03313=1068.502,111.604,426.771,172.888,27.034,154.906
C03314=1068.497,111.355,426.791,172.887,27.031,154.906
C03315=1068.488,110.979,426.820,172.885,27.027,154.905
C03316=1068.478,110.601,426.849,172.881,27.023,154.905
C03317=1068.470,110.225,426.878,172.879,27.019,154.904
C03318=1068.461,109.847,426.906,172.877,27.015,154.903
C03319=1068.455,109.598,426.926,172.875,27.013,154.903
C03320=1068.449,109.349,426.945,172.874,27.010,154.903
C03321=1068.443,109.100,426.964,172.872,27.007,154.902
C03322=1068.438,108.850,426.983,172.871,27.004,154.902
C03323=1068.432,108.601,427.003,172.870,27.001,154.902
C03324=1068.425,108.352,427.021,172.867,26.999,154.901
C03325=1068.420,108.102,427.041,172.866,26.996,154.901
C03326=1068.415,107.854,427.059,172.864,26.993,154.901
C03327=1068.409,107.605,427.079,172.863,26.990,154.900
C03328=1068.402,107.356,427.098,172.861,26.988,154.900
C03329=1068.397,107.106,427.117,172.860,26.985,154.899
C03330=1068.391,106.857,427.137,172.858,26.982,154.899
C03331=1068.385,106.607,427.156,172.857,26.980,154.899
C03332=1068.379,106.358,427.174,172.855,26.977,154.898
C03333=1068.374,106.110,427.193,172.854,26.975,154.898
C03334=1068.368,105.860,427.213,172.852,26.972,154.898
C03335=1068.362,105.611,427.231,172.851,26.969,154.897
C03336=1068.356,105.362,427.250,172.848,26.966,154.897
C03337=1068.350,105.112,427.270,172.847,26.963,154.896
C03338=1068.345,104.863,427.289,172.845,26.960,154.896
C03339=1068.339,104.614,427.307,172.844,26.958,154.896
C03340=1068.333,104.365,427.326,172.842,26.955,154.895
C03341=1068.327,104.115,427.346,172.841,26.952,154.895
C03342=1068.321,103.866,427.364,172.840,26.950,154.894
C03343=1068.316,103.618,427.383,172.838,26.947,154.894
C03344=1068.310,103.368,427.402,172.837,26.944,154.894
C03345=1068.304,103.119,427.421,172.835,26.942,154.893
C03346=1068.298,102.870,427.440,172.834,26.939,154.893
C03347=1068.293,102.621,427.459,172.832,26.936,154.893
C03348=1068.288,102.371,427.478,172.831,26.933,154.892
C03349=1068.281,102.122,427.496,172.828,26.930,154.892
C03350=1068.275,101.872,427.516,172.827,26.927,154.891
C03351=1068.266,101.468,427.546,172.825,26.923,154.891
C03352=1068.257,101.064,427.577,172.822,26.919,154.890
C03353=1068.247,100.659,427.607,172.819,26.914,154.890
C03354=1068.238,100.254,427.638,172.817,26.910,154.889
C03355=1068.231,100.005,427.657,172.816,26.907,154.889
C03356=1068.226,99.756,427.674,172.814,26.905,154.888
C03357=1068.220,99.507,427.694,172.813,26.902,154.888
C03358=1068.214,99.258,427.712,172.811,26.899,154.888
C03359=1068.208,99.008,427.732,172.810,26.897,154.887
C03360=1068.202,98.759,427.750,172.808,26.894,154.887
C03361=1068.197,98.510,427.768,172.807,26.891,154.886
C03362=1068.190,98.261,427.787,172.805,26.889,154.886
C03363=1068.185,98.011,427.806,172.803,26.886,154.886
C03364=1068.178,97.762,427.825,172.802,26.883,154.885
C03365=1068.174,97.513,427.843,172.800,26.880,154.885
C03366=1068.167,97.264,427.862,172.799,26.877,154.884
C03367=1068.161,97.014,427.880,172.797,26.875,154.884
C03368=1068.156,96.766,427.899,172.796,26.872,154.884
C03369=1068.150,96.516,427.917,172.794,26.869,154.883
C03370=1068.144,96.266,427.936,172.793,26.866,154.883
C03371=1068.137,96.017,427.955,172.791,26.864,154.883
C03372=1068.133,95.768,427.973,172.790,26.861,154.882
C03373=1068.126,95.519,427.992,172.788,26.859,154.882
C03374=1068.120,95.270,428.011,172.787,26.856,154.881
C03375=1068.113,94.987,428.031,172.785,26.853,154.881
C03376=1068.107,94.704,428.053,172.783,26.849,154.881
C03377=1068.101,94.420,428.074,172.782,26.846,154.880
C03378=1068.095,94.137,428.094,172.780,26.844,154.880
C03379=1068.088,93.888,428.113,172.779,26.841,154.879
C03380=1068.082,93.639,428.132,172.777,26.838,154.879
C03381=1068.077,93.389,428.150,172.775,26.835,154.879
C03382=1068.071,93.140,428.169,172.774,26.832,154.878
C03383=1068.065,92.890,428.187,172.772,26.829,154.878
C03384=1068.059,92.642,428.205,172.771,26.827,154.878
C03385=1068.053,92.393,428.224,172.769,26.824,154.877
C03386=1068.048,92.143,428.242,172.768,26.821,154.877
C03387=1068.042,91.894,428.261,172.766,26.818,154.876
C03388=1068.036,91.644,428.279,172.765,26.816,154.876
C03389=1068.031,91.396,428.298,172.763,26.813,154.876
C03390=1068.024,91.146,428.316,172.762,26.810,154.875
C03391=1068.019,90.897,428.335,172.760,26.808,154.875
C03392=1068.013,90.648,428.352,172.759,26.805,154.874
C03393=1068.007,90.398,428.371,172.757,26.802,154.874
C03394=1068.001,90.149,428.389,172.756,26.799,154.874
C03395=1067.995,89.900,428.407,172.754,26.797,154.873
C03396=1067.990,89.650,428.426,172.753,26.794,154.873
C03397=1067.984,89.402,428.444,172.752,26.791,154.873
C03398=1067.978,89.152,428.462,172.750,26.789,154.872
C03399=1067.971,88.902,428.480,172.749,26.786,154.872
C03400=1067.966,88.654,428.498,172.747,26.783,154.871
C03401=1067.959,88.404,428.516,172.746,26.781,154.871
C03402=1067.954,88.155,428.535,172.744,26.778,154.871
C03403=1067.948,87.906,428.553,172.743,26.776,154.870
C03404=1067.942,87.657,428.572,172.741,26.773,154.870
C03405=1067.936,87.408,428.589,172.740,26.770,154.870
C03406=1067.930,87.158,428.607,172.738,26.767,154.869
C03407=1067.924,86.909,428.626,172.737,26.764,154.869
C03408=1067.918,86.660,428.643,172.735,26.762,154.868
C03409=1067.913,86.410,428.662,172.734,26.759,154.868
C03410=1067.907,86.161,428.680,172.733,26.756,154.868
C03411=1067.901,85.911,428.698,172.731,26.753,154.867
C03412=1067.895,85.662,428.716,172.729,26.751,154.867
C03413=1067.889,85.413,428.734,172.727,26.748,154.867
C03414=1067.883,85.164,428.752,172.726,26.745,154.866
C03415=1067.877,84.914,428.770,172.724,26.742,154.866
C03416=1067.871,84.665,428.788,172.723,26.740,154.865
C03417=1067.866,84.416,428.807,172.721,26.737,154.865
C03418=1067.860,84.166,428.824,172.720,26.735,154.865
C03419=1067.854,83.918,428.843,172.718,26.732,154.864
C03420=1067.848,83.668,428.861,172.717,26.729,154.864
C03421=1067.842,83.418,428.879,172.716,26.726,154.864
C03422=1067.836,83.169,428.896,172.714,26.724,154.863
C03423=1067.830,82.920,428.915,172.713,26.721,154.863
C03424=1067.825,82.671,428.932,172.711,26.718,154.862
C03425=1067.818,82.421,428.950,172.710,26.715,154.862
C03426=1067.813,82.172,428.968,172.708,26.712,154.862
C03427=1067.807,81.922,428.986,172.707,26.710,154.861
C03428=1067.802,81.674,429.005,172.705,26.707,154.861
C03429=1067.796,81.424,429.023,172.704,26.704,154.861
C03430=1067.790,81.175,429.040,172.702,26.702,154.860
C03431=1067.784,80.925,429.058,172.701,26.699,154.860
C03432=1067.778,80.676,429.076,172.700,26.696,154.859
C03433=1067.773,80.428,429.094,172.698,26.693,154.859
C03434=1067.766,80.178,429.112,172.697,26.690,154.859
C03435=1067.761,79.929,429.129,172.695,26.688,154.858
C03436=1067.755,79.679,429.147,172.694,26.685,154.858
C03437=1067.749,79.430,429.165,172.692,26.682,154.857
C03438=1067.743,79.181,429.183,172.691,26.680,154.857
C03439=1067.737,78.897,429.204,172.689,26.677,154.857
C03440=1067.730,78.614,429.224,172.688,26.673,154.856
C03441=1067.724,78.332,429.244,172.686,26.670,154.856
C03442=1067.717,78.049,429.264,172.684,26.667,154.855
C03443=1067.711,77.799,429.282,172.683,26.665,154.855
C03444=1067.705,77.550,429.299,172.681,26.662,154.855
C03445=1067.699,77.300,429.317,172.680,26.659,154.854
C03446=1067.693,77.051,429.335,172.679,26.657,154.854
C03447=1067.687,76.802,429.353,172.677,26.654,154.854
C03448=1067.682,76.553,429.370,172.676,26.651,154.853
C03449=1067.675,76.303,429.388,172.674,26.648,154.853
C03450=1067.669,76.054,429.405,172.673,26.646,154.852
C03451=1067.664,75.805,429.423,172.671,26.643,154.852
C03452=1067.658,75.555,429.441,172.670,26.640,154.852
C03453=1067.652,75.306,429.458,172.668,26.637,154.851
C03454=1067.646,75.057,429.476,172.667,26.635,154.851
C03455=1067.640,74.808,429.493,172.665,26.632,154.851
C03456=1067.634,74.558,429.511,172.664,26.629,154.850
C03457=1067.628,74.309,429.529,172.663,26.626,154.850
C03458=1067.623,74.060,429.546,172.661,26.624,154.849
C03459=1067.617,73.810,429.564,172.660,26.621,154.849
C03460=1067.611,73.561,429.582,172.658,26.619,154.849
C03461=1067.604,73.312,429.599,172.657,26.616,154.848
C03462=1067.599,73.063,429.617,172.655,26.613,154.848
C03463=1067.594,72.813,429.634,172.654,26.610,154.847
C03464=1067.587,72.563,429.652,172.652,26.608,154.847
C03465=1067.582,72.314,429.669,172.651,26.605,154.847
C03466=1067.575,72.065,429.687,172.650,26.602,154.846
C03467=1067.570,71.816,429.704,172.648,26.599,154.846
C03468=1067.564,71.567,429.722,172.647,26.596,154.846
C03469=1067.558,71.317,429.740,172.645,26.594,154.845
C03470=1067.552,71.068,429.757,172.644,26.591,154.845
C03471=1067.546,70.818,429.774,172.642,26.588,154.845
C03472=1067.540,70.569,429.791,172.641,26.586,154.844
C03473=1067.535,70.320,429.809,172.640,26.583,154.844
C03474=1067.529,70.070,429.827,172.638,26.580,154.843
C03475=1067.522,69.821,429.844,172.637,26.578,154.843
C03476=1067.517,69.572,429.861,172.635,26.575,154.843
C03477=1067.511,69.322,429.879,172.634,26.572,154.842
C03478=1067.505,69.073,429.896,172.632,26.569,154.842
C03479=1067.499,68.824,429.913,172.631,26.567,154.842
C03480=1067.493,68.575,429.931,172.629,26.564,154.841
C03481=1067.487,68.325,429.947,172.628,26.561,154.841
C03482=1067.482,68.076,429.965,172.626,26.558,154.840
C03483=1067.476,67.826,429.983,172.625,26.556,154.840
C03484=1067.469,67.578,430.000,172.624,26.553,154.840
C03485=1067.464,67.328,430.017,172.622,26.550,154.839
C03486=1067.458,67.078,430.035,172.621,26.547,154.839
C03487=1067.452,66.830,430.052,172.619,26.545,154.839
C03488=1067.447,66.580,430.068,172.618,26.542,154.838
C03489=1067.440,66.330,430.086,172.616,26.540,154.838
C03490=1067.434,66.081,430.103,172.615,26.537,154.837
C03491=1067.429,65.832,430.120,172.614,26.534,154.837
C03492=1067.422,65.582,430.137,172.612,26.532,154.837
C03493=1067.417,65.333,430.155,172.611,26.529,154.836
C03494=1067.411,65.084,430.171,172.609,26.526,154.836
C03495=1067.404,64.834,430.189,172.608,26.523,154.836
C03496=1067.398,64.585,430.206,172.606,26.521,154.835
C03497=1067.393,64.336,430.223,172.605,26.518,154.835
C03498=1067.386,64.086,430.240,172.603,26.515,154.834
C03499=1067.381,63.837,430.258,172.602,26.513,154.834
C03500=1067.375,63.588,430.274,172.600,26.510,154.834
C03501=1067.369,63.338,430.292,172.599,26.507,154.833
C03502=1067.363,63.089,430.308,172.597,26.505,154.833
C03503=1067.356,62.806,430.328,172.596,26.501,154.833
C03504=1067.349,62.522,430.348,172.595,26.498,154.832
C03505=1067.342,62.240,430.366,172.593,26.496,154.832
C03506=1067.335,61.956,430.386,172.591,26.493,154.831
C03507=1067.329,61.707,430.403,172.590,26.490,154.831
C03508=1067.323,61.457,430.420,172.588,26.487,154.831
C03509=1067.317,61.208,430.437,172.587,26.485,154.830
C03510=1067.311,60.959,430.454,172.585,26.482,154.830
C03511=1067.305,60.709,430.471,172.585,26.479,154.830
C03512=1067.299,60.460,430.487,172.583,26.477,154.829
C03513=1067.293,60.211,430.505,172.582,26.474,154.829
C03514=1067.287,59.962,430.521,172.580,26.471,154.828
C03515=1067.280,59.712,430.538,172.579,26.469,154.828
C03516=1067.275,59.463,430.555,172.577,26.466,154.828
C03517=1067.269,59.214,430.572,172.576,26.463,154.827
C03518=1067.263,58.964,430.588,172.575,26.461,154.827
C03519=1067.257,58.714,430.606,172.573,26.458,154.827
C03520=1067.251,58.465,430.623,172.572,26.455,154.826
C03521=1067.245,58.216,430.639,172.570,26.453,154.826
C03522=1067.239,57.967,430.656,172.569,26.450,154.826
C03523=1067.233,57.717,430.673,172.567,26.447,154.825
C03524=1067.226,57.468,430.690,172.566,26.444,154.825
C03525=1067.221,57.219,430.707,172.564,26.442,154.825
C03526=1067.215,56.969,430.723,172.563,26.439,154.824
C03527=1067.208,56.720,430.740,172.562,26.436,154.824
C03528=1067.203,56.470,430.757,172.560,26.434,154.823
C03529=1067.197,56.221,430.774,172.559,26.431,154.823
C03530=1067.191,55.972,430.791,172.557,26.428,154.823
C03531=1067.186,55.722,430.807,172.556,26.425,154.822
C03532=1067.179,55.472,430.824,172.554,26.423,154.822
C03533=1067.173,55.224,430.841,172.553,26.420,154.822
C03534=1067.167,54.974,430.857,172.552,26.417,154.821
C03535=1067.162,54.725,430.874,172.550,26.415,154.821
C03536=1067.156,54.476,430.891,172.549,26.412,154.821
C03537=1067.150,54.227,430.907,172.547,26.409,154.820
C03538=1067.144,53.976,430.925,172.546,26.407,154.820
C03539=1067.138,53.727,430.941,172.544,26.404,154.819
C03540=1067.132,53.478,430.958,172.543,26.401,154.819
C03541=1067.126,53.229,430.974,172.541,26.399,154.819
C03542=1067.120,52.979,430.991,172.540,26.396,154.818
C03543=1067.114,52.730,431.008,172.539,26.393,154.818
C03544=1067.108,52.481,431.024,172.537,26.391,154.818
C03545=1067.102,52.231,431.041,172.536,26.388,154.817
C03546=1067.096,51.981,431.058,172.534,26.385,154.817
C03547=1067.090,51.733,431.075,172.533,26.383,154.817
C03548=1067.084,51.483,431.091,172.531,26.380,154.816
C03549=1067.079,51.234,431.108,172.530,26.377,154.816
C03550=1067.073,50.984,431.124,172.529,26.374,154.815
C03551=1067.067,50.735,431.140,172.528,26.372,154.815
C03552=1067.061,50.486,431.157,172.527,26.369,154.815
C03553=1067.055,50.237,431.173,172.525,26.366,154.814
C03554=1067.049,49.986,431.191,172.524,26.363,154.814
C03555=1067.043,49.737,431.207,172.522,26.361,154.814
C03556=1067.037,49.488,431.223,172.521,26.358,154.813
C03557=1067.031,49.238,431.239,172.519,26.355,154.813
C03558=1067.026,48.989,431.256,172.518,26.353,154.812
C03559=1067.020,48.740,431.273,172.517,26.350,154.812
C03560=1067.014,48.491,431.289,172.515,26.347,154.812
C03561=1067.008,48.241,431.306,172.514,26.345,154.811
C03562=1067.003,47.992,431.323,172.512,26.342,154.811
C03563=1066.997,47.742,431.339,172.511,26.339,154.810
C03564=1066.991,47.493,431.355,172.509,26.337,154.810
C03565=1066.985,47.244,431.371,172.508,26.334,154.810
C03566=1066.979,46.994,431.388,172.507,26.331,154.809
C03567=1066.972,46.711,431.407,172.505,26.328,154.809
C03568=1066.966,46.427,431.425,172.504,26.325,154.809
C03569=1066.959,46.144,431.444,172.502,26.321,154.808
C03570=1066.953,45.860,431.462,172.500,26.319,154.808
C03571=1066.947,45.611,431.478,172.499,26.316,154.807
C03572=1066.942,45.361,431.495,172.497,26.313,154.807
C03573=1066.936,45.112,431.512,172.496,26.311,154.807
C03574=1066.930,44.863,431.528,172.495,26.308,154.806
C03575=1066.924,44.613,431.544,172.493,26.305,154.806
C03576=1066.918,44.364,431.560,172.492,26.302,154.805
C03577=1066.913,44.114,431.577,172.490,26.299,154.805
C03578=1066.907,43.865,431.593,172.489,26.297,154.805
C03579=1066.901,43.616,431.610,172.487,26.294,154.804
C03580=1066.895,43.366,431.626,172.486,26.291,154.804
C03581=1066.889,43.117,431.642,172.485,26.289,154.804
C03582=1066.883,42.868,431.658,172.484,26.286,154.803
C03583=1066.877,42.618,431.675,172.483,26.283,154.803
C03584=1066.871,42.369,431.691,172.481,26.280,154.803
C03585=1066.865,42.120,431.707,172.480,26.278,154.802
C03586=1066.859,41.870,431.723,172.478,26.275,154.802
C03587=1066.853,41.621,431.740,172.477,26.272,154.801
C03588=1066.847,41.371,431.755,172.475,26.270,154.801
C03589=1066.841,41.122,431.772,172.474,26.267,154.801
C03590=1066.835,40.872,431.788,172.473,26.264,154.800
C03591=1066.829,40.623,431.803,172.471,26.262,154.800
C03592=1066.823,40.374,431.820,172.470,26.259,154.800
C03593=1066.817,40.125,431.836,172.468,26.256,154.799
C03594=1066.811,39.875,431.852,172.467,26.254,154.799
C03595=1066.805,39.625,431.868,172.465,26.251,154.799
C03596=1066.799,39.376,431.884,172.464,26.248,154.798
C03597=1066.793,39.127,431.900,172.463,26.245,154.798
C03598=1066.787,38.877,431.917,172.461,26.243,154.798
C03599=1066.781,38.628,431.933,172.460,26.240,154.797
C03600=1066.776,38.378,431.948,172.458,26.237,154.797
C03601=1066.770,38.128,431.965,172.457,26.235,154.797
C03602=1066.764,37.879,431.981,172.456,26.232,154.796
C03603=1066.758,37.630,431.997,172.454,26.229,154.796
C03604=1066.752,37.380,432.012,172.453,26.227,154.795
C03605=1066.746,37.131,432.028,172.451,26.224,154.795
C03606=1066.740,36.881,432.045,172.450,26.222,154.795
C03607=1066.734,36.632,432.061,172.448,26.219,154.794
C03608=1066.728,36.382,432.076,172.447,26.216,154.794
C03609=1066.721,36.133,432.092,172.446,26.214,154.794
C03610=1066.715,35.884,432.108,172.445,26.211,154.793
C03611=1066.710,35.634,432.125,172.443,26.209,154.793
C03612=1066.704,35.384,432.140,172.442,26.206,154.793
C03613=1066.698,35.136,432.155,172.441,26.203,154.792
C03614=1066.692,34.887,432.172,172.439,26.201,154.792
C03615=1066.686,34.637,432.187,172.438,26.198,154.792
C03616=1066.680,34.387,432.203,172.436,26.195,154.791
C03617=1066.674,34.138,432.219,172.435,26.193,154.791
C03618=1066.668,33.888,432.235,172.434,26.190,154.790
C03619=1066.662,33.639,432.251,172.432,26.188,154.790
C03620=1066.656,33.389,432.266,172.431,26.185,154.790
C03621=1066.650,33.140,432.282,172.429,26.182,154.789
C03622=1066.644,32.891,432.298,172.428,26.180,154.789
C03623=1066.638,32.641,432.314,172.426,26.177,154.789
C03624=1066.632,32.392,432.329,172.425,26.174,154.788
C03625=1066.626,32.142,432.345,172.423,26.172,154.788
C03626=1066.620,31.893,432.361,172.422,26.169,154.788
C03627=1066.614,31.644,432.377,172.421,26.166,154.787
C03628=1066.608,31.394,432.392,172.419,26.164,154.787
C03629=1066.602,31.145,432.408,172.418,26.161,154.787
C03630=1066.596,30.895,432.424,172.416,26.158,154.786
C03631=1066.590,30.612,432.442,172.415,26.156,154.786
C03632=1066.583,30.328,432.459,172.414,26.153,154.786
C03633=1066.576,30.045,432.477,172.412,26.149,154.785
C03634=1066.569,29.761,432.495,172.410,26.146,154.785
C03635=1066.563,29.512,432.511,172.408,26.144,154.784
C03636=1066.558,29.262,432.527,172.407,26.141,154.784
C03637=1066.552,29.014,432.542,172.406,26.138,154.784
C03638=1066.546,28.764,432.558,172.405,26.136,154.783
C03639=1066.540,28.514,432.573,172.404,26.133,154.783
C03640=1066.534,28.265,432.589,172.402,26.131,154.783
C03641=1066.528,28.015,432.604,172.401,26.128,154.782
